LIN {X 0,Y 365.987,Z 762.314,A -85,B 0,C 180,E1 17582.28,E2 17582.28} C_VEL
LIN {X 0,Y 362.465,Z 777.838,A -85,B 0,C 180,E1 17579.586,E2 17579.586} C_VEL
LIN {X 0,Y 359.456,Z 791.622,A -85,B 0,C 180,E1 17576.759,E2 17576.759} C_VEL
LIN {X 0,Y 356.962,Z 803.911,A -85,B 0,C 180,E1 17573.786,E2 17573.786} C_VEL
LIN {X 0,Y 354.994,Z 814.892,A -85,B 0,C 180,E1 17570.612,E2 17570.612} C_VEL
LIN {X 0,Y 353.626,Z 823.927,A -85,B 0,C 180,E1 17567.438,E2 17567.438} C_VEL
LIN {X 0,Y 352.73,Z 831.669,A -85,B 0,C 180,E1 17564.108,E2 17564.108} C_VEL
LIN {X 0,Y 352.306,Z 837.449,A -85,B 0,C 180,E1 17560.895,E2 17560.895} C_VEL
LIN {X 0,Y 352.156,Z 841.876,A -85,B 0,C 180,E1 17557.503,E2 17557.503} C_VEL
LIN {X 0,Y 352.166,Z 844.497,A -85,B 0,C 180,E1 17554.395,E2 17554.395} C_VEL
LIN {X 0,Y 352.213,Z 845.642,A -85,B 0,C 180,E1 17551.137,E2 17551.137} C_VEL
LIN {X 0,Y 352.217,Z 845.355,A -85,B 0,C 180,E1 17548.046,E2 17548.046} C_VEL
LIN {X 0,Y 352.206,Z 843.421,A -85,B 0,C 180,E1 17544.786,E2 17544.786} C_VEL
LIN {X 0,Y 352.225,Z 839.976,A -85,B 0,C 180,E1 17541.51,E2 17541.51} C_VEL
LIN {X 0,Y 352.423,Z 835.044,A -85,B 0,C 180,E1 17538.378,E2 17538.378} C_VEL
LIN {X 0,Y 352.934,Z 828.184,A -85,B 0,C 180,E1 17535.031,E2 17535.031} C_VEL
LIN {X 0,Y 353.839,Z 820.007,A -85,B 0,C 180,E1 17531.889,E2 17531.889} C_VEL
LIN {X 0,Y 355.279,Z 809.812,A -85,B 0,C 180,E1 17528.677,E2 17528.677} C_VEL
LIN {X 0,Y 357.273,Z 797.828,A -85,B 0,C 180,E1 17525.53,E2 17525.53} C_VEL
LIN {X 0,Y 359.648,Z 784.987,A -85,B 0,C 180,E1 17522.694,E2 17522.694} C_VEL
LIN {X 0,Y 362.722,Z 769.51,A -85,B 0,C 180,E1 17519.795,E2 17519.795} C_VEL
LIN {X 0,Y 366.339,Z 752.001,A -85,B 0,C 180,E1 17517.031,E2 17517.031} C_VEL
LIN {X 0,Y 369.994,Z 734.378,A -85,B 0,C 180,E1 17514.667,E2 17514.667} C_VEL
LIN {X 0,Y 373.861,Z 715.366,A -85,B 0,C 180,E1 17512.523,E2 17512.523} C_VEL
LIN {X 0,Y 377.906,Z 695.003,A -85,B 0,C 180,E1 17510.58,E2 17510.58} C_VEL
LIN {X 0,Y 382.09,Z 673.141,A -85,B 0,C 180,E1 17508.841,E2 17508.841} C_VEL
LIN {X 0,Y 386.129,Z 650.609,A -85,B 0,C 180,E1 17507.368,E2 17507.368} C_VEL
LIN {X 0,Y 390.147,Z 626.368,A -85,B 0,C 180,E1 17506.112,E2 17506.112} C_VEL
LIN {X 0,Y 393.895,Z 600.938,A -85,B 0,C 180,E1 17505.107,E2 17505.107} C_VEL
LIN {X 0,Y 396.97,Z 573.317,A -85,B 0,C 180,E1 17504.265,E2 17504.265} C_VEL
LIN {X 0,Y 403.928,Z 504.871,A -85,B 0,C 180,E1 17502.414,E2 17502.414} C_VEL
LIN {X 0,Y 412.99,Z 436.759,A -85,B 0,C 180,E1 17500.479,E2 17500.479} C_VEL
LIN {X 0,Y 424.745,Z 366.791,A -85,B 0,C 180,E1 17498.462,E2 17498.462} C_VEL
LIN {X 0,Y 426.24,Z 358.784,A -85,B 0,C 180,E1 17498.201,E2 17498.201} C_VEL
LIN {X 0,Y 426.55,Z 354.223,A -85,B 0,C 180,E1 17497.156,E2 17497.156} C_VEL
LIN {X 0,Y 427.054,Z 351.949,A -85,B 0,C 180,E1 17496.325,E2 17496.325} C_VEL
LIN {X 0,Y 427.299,Z 351.738,A -85,B 0,C 180,E1 17495.886,E2 17495.886} C_VEL
LIN {X 0,Y 427.284,Z 352.228,A -85,B 0,C 180,E1 17495.743,E2 17495.743} C_VEL
LIN {X 0,Y 415.748,Z 415.551,A -85,B 0,C 180,E1 17493.926,E2 17493.926} C_VEL
LIN {X 0,Y 406.562,Z 477.379,A -85,B 0,C 180,E1 17492.151,E2 17492.151} C_VEL
LIN {X 0,Y 399.106,Z 542.752,A -85,B 0,C 180,E1 17490.336,E2 17490.336} C_VEL
LIN {X 0,Y 396.477,Z 567.509,A -85,B 0,C 180,E1 17489.494,E2 17489.494} C_VEL
LIN {X 0,Y 393.293,Z 591.201,A -85,B 0,C 180,E1 17488.387,E2 17488.387} C_VEL
LIN {X 0,Y 389.623,Z 613.913,A -85,B 0,C 180,E1 17487.016,E2 17487.016} C_VEL
LIN {X 0,Y 385.453,Z 636.079,A -85,B 0,C 180,E1 17485.343,E2 17485.343} C_VEL
LIN {X 0,Y 381.122,Z 656.641,A -85,B 0,C 180,E1 17483.421,E2 17483.421} C_VEL
LIN {X 0,Y 376.79,Z 675.215,A -85,B 0,C 180,E1 17481.32,E2 17481.32} C_VEL
LIN {X 0,Y 372.567,Z 692.109,A -85,B 0,C 180,E1 17479.032,E2 17479.032} C_VEL
LIN {X 0,Y 368.567,Z 707.5,A -85,B 0,C 180,E1 17476.551,E2 17476.551} C_VEL
LIN {X 0,Y 364.962,Z 721.167,A -85,B 0,C 180,E1 17473.953,E2 17473.953} C_VEL
LIN {X 0,Y 361.517,Z 734.047,A -85,B 0,C 180,E1 17471.003,E2 17471.003} C_VEL
LIN {X 0,Y 358.694,Z 744.9,A -85,B 0,C 180,E1 17468.014,E2 17468.014} C_VEL
LIN {X 0,Y 356.397,Z 754.518,A -85,B 0,C 180,E1 17464.83,E2 17464.83} C_VEL
LIN {X 0,Y 354.639,Z 762.753,A -85,B 0,C 180,E1 17461.456,E2 17461.456} C_VEL
LIN {X 0,Y 353.45,Z 769.171,A -85,B 0,C 180,E1 17458.057,E2 17458.057} C_VEL
LIN {X 0,Y 352.739,Z 774.193,A -85,B 0,C 180,E1 17454.472,E2 17454.472} C_VEL
LIN {X 0,Y 352.395,Z 777.476,A -85,B 0,C 180,E1 17451.025,E2 17451.025} C_VEL
LIN {X 0,Y 352.253,Z 779.104,A -85,B 0,C 180,E1 17447.711,E2 17447.711} C_VEL
LIN {X 0,Y 352.227,Z 779.342,A -85,B 0,C 180,E1 17444.223,E2 17444.223} C_VEL
LIN {X 0,Y 352.257,Z 778.2,A -85,B 0,C 180,E1 17440.946,E2 17440.946} C_VEL
LIN {X 0,Y 352.388,Z 775.578,A -85,B 0,C 180,E1 17437.656,E2 17437.656} C_VEL
LIN {X 0,Y 352.757,Z 771.52,A -85,B 0,C 180,E1 17434.303,E2 17434.303} C_VEL
LIN {X 0,Y 353.475,Z 765.83,A -85,B 0,C 180,E1 17430.935,E2 17430.935} C_VEL
LIN {X 0,Y 354.654,Z 758.568,A -85,B 0,C 180,E1 17427.615,E2 17427.615} C_VEL
LIN {X 0,Y 356.419,Z 749.576,A -85,B 0,C 180,E1 17424.307,E2 17424.307} C_VEL
LIN {X 0,Y 358.837,Z 738.627,A -85,B 0,C 180,E1 17421.025,E2 17421.025} C_VEL
LIN {X 0,Y 361.659,Z 726.557,A -85,B 0,C 180,E1 17418.048,E2 17418.048} C_VEL
LIN {X 0,Y 365.008,Z 712.783,A -85,B 0,C 180,E1 17415.193,E2 17415.193} C_VEL
LIN {X 0,Y 368.625,Z 698.003,A -85,B 0,C 180,E1 17412.603,E2 17412.603} C_VEL
LIN {X 0,Y 372.462,Z 681.884,A -85,B 0,C 180,E1 17410.231,E2 17410.231} C_VEL
LIN {X 0,Y 376.443,Z 664.226,A -85,B 0,C 180,E1 17408.041,E2 17408.041} C_VEL
LIN {X 0,Y 380.473,Z 645.175,A -85,B 0,C 180,E1 17406.063,E2 17406.063} C_VEL
LIN {X 0,Y 384.229,Z 625.745,A -85,B 0,C 180,E1 17404.382,E2 17404.382} C_VEL
LIN {X 0,Y 387.547,Z 605.931,A -85,B 0,C 180,E1 17402.983,E2 17402.983} C_VEL
LIN {X 0,Y 390.527,Z 585.074,A -85,B 0,C 180,E1 17401.793,E2 17401.793} C_VEL
LIN {X 0,Y 393.119,Z 563.144,A -85,B 0,C 180,E1 17400.816,E2 17400.816} C_VEL
LIN {X 0,Y 395.064,Z 541.461,A -85,B 0,C 180,E1 17400.105,E2 17400.105} C_VEL
LIN {X 0,Y 397.486,Z 497.686,A -85,B 0,C 180,E1 17399.14,E2 17399.14} C_VEL
LIN {X 0,Y 405.981,Z 342.64,A -85,B 0,C 180,E1 17395.845,E2 17395.845} C_VEL
LIN {X 0,Y 392.058,Z 321.721,A -85,B 0,C 180,E1 17393.047,E2 17393.047} C_VEL
LIN {X 0,Y 379.817,Z 304.351,A -85,B 0,C 180,E1 17390.335,E2 17390.335} C_VEL
LIN {X 0,Y 369.449,Z 290.34,A -85,B 0,C 180,E1 17387.849,E2 17387.849} C_VEL
LIN {X 0,Y 365.575,Z 285.201,A -85,B 0,C 180,E1 17386.854,E2 17386.854} C_VEL
LIN {X 0,Y 362.474,Z 280.851,A -85,B 0,C 180,E1 17386.034,E2 17386.034} C_VEL
LIN {X 0,Y 358.985,Z 276.815,A -85,B 0,C 180,E1 17385.117,E2 17385.117} C_VEL
LIN {X 0,Y 357.684,Z 274.526,A -85,B 0,C 180,E1 17384.73,E2 17384.73} C_VEL
LIN {X 0,Y 355.038,Z 271.984,A -85,B 0,C 180,E1 17384.017,E2 17384.017} C_VEL
LIN {X 0,Y 353.876,Z 268.895,A -85,B 0,C 180,E1 17383.606,E2 17383.606} C_VEL
LIN {X 0,Y 353.84,Z 268.66,A -85,B 0,C 180,E1 17379.557,E2 17379.557} C_VEL
LIN {X 0,Y 353.836,Z 268.649,A -85,B 0,C 180,E1 17375.515,E2 17375.515} C_VEL
LIN {X 0,Y 353.842,Z 268.652,A -85,B 0,C 180,E1 17371.297,E2 17371.297} C_VEL
LIN {X 0,Y 353.839,Z 268.655,A -85,B 0,C 180,E1 17367.248,E2 17367.248} C_VEL
LIN {X 0,Y 353.825,Z 268.656,A -85,B 0,C 180,E1 17363.609,E2 17363.609} C_VEL
LIN {X 0,Y 352.854,Z 268.776,A -85,B 0,C 180,E1 17362.362,E2 17362.362} C_VEL
LIN {X 0,Y 348.27,Z 269.351,A -85,B 0,C 180,E1 17360.005,E2 17360.005} C_VEL
LIN {X 0,Y 346.039,Z 269.618,A -85,B 0,C 180,E1 17358.378,E2 17358.378} C_VEL
LIN {X 0,Y 345.889,Z 269.637,A -85,B 0,C 180,E1 17357.915,E2 17357.915} C_VEL
LIN {X 0,Y 345.884,Z 269.641,A -85,B 0,C 180,E1 17353.67,E2 17353.67} C_VEL
LIN {X 0,Y 345.884,Z 269.643,A -85,B 0,C 180,E1 17349.351,E2 17349.351} C_VEL
LIN {X 0,Y 345.884,Z 269.643,A -85,B 0,C 180,E1 17345.18,E2 17345.18} C_VEL
LIN {X 0,Y 345.882,Z 269.642,A -85,B 0,C 180,E1 17341.137,E2 17341.137} C_VEL
LIN {X 0,Y 345.885,Z 269.64,A -85,B 0,C 180,E1 17336.956,E2 17336.956} C_VEL
LIN {X 0,Y 345.885,Z 269.639,A -85,B 0,C 180,E1 17332.834,E2 17332.834} C_VEL
LIN {X 0,Y 345.887,Z 269.642,A -85,B 0,C 180,E1 17328.723,E2 17328.723} C_VEL
LIN {X 0,Y 345.888,Z 269.645,A -85,B 0,C 180,E1 17324.618,E2 17324.618} C_VEL
LIN {X 0,Y 345.901,Z 269.645,A -85,B 0,C 180,E1 17320.349,E2 17320.349} C_VEL
LIN {X 0,Y 345.903,Z 269.647,A -85,B 0,C 180,E1 17316.13,E2 17316.13} C_VEL
LIN {X 0,Y 345.9,Z 269.648,A -85,B 0,C 180,E1 17311.811,E2 17311.811} C_VEL
LIN {X 0,Y 345.902,Z 269.65,A -85,B 0,C 180,E1 17307.732,E2 17307.732} C_VEL
LIN {X 0,Y 345.886,Z 269.652,A -85,B 0,C 180,E1 17303.508,E2 17303.508} C_VEL
LIN {X 0,Y 345.883,Z 269.651,A -85,B 0,C 180,E1 17299.414,E2 17299.414} C_VEL
LIN {X 0,Y 345.875,Z 269.649,A -85,B 0,C 180,E1 17295.249,E2 17295.249} C_VEL
LIN {X 0,Y 345.87,Z 269.645,A -85,B 0,C 180,E1 17291.165,E2 17291.165} C_VEL
LIN {X 0,Y 345.861,Z 269.646,A -85,B 0,C 180,E1 17286.972,E2 17286.972} C_VEL
LIN {X 0,Y 345.859,Z 269.653,A -85,B 0,C 180,E1 17282.815,E2 17282.815} C_VEL
LIN {X 0,Y 345.856,Z 269.654,A -85,B 0,C 180,E1 17278.507,E2 17278.507} C_VEL
LIN {X 0,Y 345.859,Z 269.645,A -85,B 0,C 180,E1 17274.357,E2 17274.357} C_VEL
LIN {X 0,Y 345.863,Z 269.654,A -85,B 0,C 180,E1 17270.177,E2 17270.177} C_VEL
LIN {X 0,Y 345.869,Z 269.645,A -85,B 0,C 180,E1 17265.944,E2 17265.944} C_VEL
LIN {X 0,Y 345.874,Z 269.647,A -85,B 0,C 180,E1 17261.806,E2 17261.806} C_VEL
LIN {X 0,Y 345.88,Z 269.65,A -85,B 0,C 180,E1 17257.669,E2 17257.669} C_VEL
LIN {X 0,Y 345.94,Z 269.93,A -85,B 0,C 180,E1 17257.391,E2 17257.391} C_VEL
LIN {X 0,Y 347.396,Z 273.438,A -85,B 0,C 180,E1 17256.416,E2 17256.416} C_VEL
LIN {X 0,Y 348.675,Z 275.305,A -85,B 0,C 180,E1 17255.789,E2 17255.789} C_VEL
LIN {X 0,Y 350.72,Z 279.095,A -85,B 0,C 180,E1 17254.681,E2 17254.681} C_VEL
LIN {X 0,Y 354.332,Z 286.186,A -85,B 0,C 180,E1 17252.727,E2 17252.727} C_VEL
LIN {X 0,Y 360.76,Z 295.311,A -85,B 0,C 180,E1 17250.803,E2 17250.803} C_VEL
LIN {X 0,Y 373.143,Z 313.414,A -85,B 0,C 180,E1 17247.524,E2 17247.524} C_VEL
LIN {X 0,Y 384.602,Z 331.118,A -85,B 0,C 180,E1 17244.772,E2 17244.772} C_VEL
LIN {X 0,Y 397.375,Z 351.926,A -85,B 0,C 180,E1 17241.964,E2 17241.964} C_VEL
LIN {X 0,Y 402.124,Z 360.571,A -85,B 0,C 180,E1 17240.95,E2 17240.95} C_VEL
LIN {X 0,Y 390.839,Z 551.737,A -85,B 0,C 180,E1 17236.825,E2 17236.825} C_VEL
LIN {X 0,Y 387.902,Z 601.626,A -85,B 0,C 180,E1 17235.696,E2 17235.696} C_VEL
LIN {X 0,Y 385.427,Z 624.723,A -85,B 0,C 180,E1 17234.955,E2 17234.955} C_VEL
LIN {X 0,Y 382.332,Z 646.717,A -85,B 0,C 180,E1 17233.981,E2 17233.981} C_VEL
LIN {X 0,Y 378.753,Z 668.624,A -85,B 0,C 180,E1 17232.72,E2 17232.72} C_VEL
LIN {X 0,Y 374.834,Z 689.594,A -85,B 0,C 180,E1 17231.211,E2 17231.211} C_VEL
LIN {X 0,Y 370.706,Z 709.59,A -85,B 0,C 180,E1 17229.456,E2 17229.456} C_VEL
LIN {X 0,Y 366.414,Z 728.906,A -85,B 0,C 180,E1 17227.391,E2 17227.391} C_VEL
LIN {X 0,Y 362.411,Z 746.037,A -85,B 0,C 180,E1 17225.21,E2 17225.21} C_VEL
LIN {X 0,Y 358.517,Z 762.431,A -85,B 0,C 180,E1 17222.752,E2 17222.752} C_VEL
LIN {X 0,Y 354.962,Z 777.449,A -85,B 0,C 180,E1 17220.09,E2 17220.09} C_VEL
LIN {X 0,Y 351.773,Z 791.358,A -85,B 0,C 180,E1 17217.168,E2 17217.168} C_VEL
LIN {X 0,Y 349.042,Z 804.226,A -85,B 0,C 180,E1 17213.962,E2 17213.962} C_VEL
LIN {X 0,Y 347.041,Z 815.018,A -85,B 0,C 180,E1 17210.753,E2 17210.753} C_VEL
LIN {X 0,Y 345.579,Z 824.337,A -85,B 0,C 180,E1 17207.336,E2 17207.336} C_VEL
LIN {X 0,Y 344.698,Z 831.806,A -85,B 0,C 180,E1 17203.929,E2 17203.929} C_VEL
LIN {X 0,Y 344.289,Z 837.602,A -85,B 0,C 180,E1 17200.54,E2 17200.54} C_VEL
LIN {X 0,Y 344.183,Z 841.606,A -85,B 0,C 180,E1 17197.174,E2 17197.174} C_VEL
LIN {X 0,Y 344.204,Z 844.093,A -85,B 0,C 180,E1 17193.829,E2 17193.829} C_VEL
LIN {X 0,Y 344.25,Z 844.918,A -85,B 0,C 180,E1 17190.83,E2 17190.83} C_VEL
LIN {X 0,Y 344.248,Z 844.467,A -85,B 0,C 180,E1 17187.64,E2 17187.64} C_VEL
LIN {X 0,Y 344.231,Z 842.486,A -85,B 0,C 180,E1 17184.498,E2 17184.498} C_VEL
LIN {X 0,Y 344.252,Z 838.914,A -85,B 0,C 180,E1 17181.143,E2 17181.143} C_VEL
LIN {X 0,Y 344.481,Z 833.899,A -85,B 0,C 180,E1 17177.936,E2 17177.936} C_VEL
LIN {X 0,Y 345.05,Z 826.928,A -85,B 0,C 180,E1 17174.537,E2 17174.537} C_VEL
LIN {X 0,Y 346.051,Z 818.588,A -85,B 0,C 180,E1 17171.292,E2 17171.292} C_VEL
LIN {X 0,Y 347.606,Z 808.312,A -85,B 0,C 180,E1 17168.04,E2 17168.04} C_VEL
LIN {X 0,Y 349.803,Z 796.062,A -85,B 0,C 180,E1 17164.791,E2 17164.791} C_VEL
LIN {X 0,Y 352.544,Z 782.277,A -85,B 0,C 180,E1 17161.728,E2 17161.728} C_VEL
LIN {X 0,Y 355.894,Z 766.369,A -85,B 0,C 180,E1 17158.763,E2 17158.763} C_VEL
LIN {X 0,Y 359.691,Z 748.99,A -85,B 0,C 180,E1 17156.03,E2 17156.03} C_VEL
LIN {X 0,Y 363.773,Z 730.564,A -85,B 0,C 180,E1 17153.579,E2 17153.579} C_VEL
LIN {X 0,Y 367.934,Z 711.368,A -85,B 0,C 180,E1 17151.414,E2 17151.414} C_VEL
LIN {X 0,Y 372.301,Z 690.641,A -85,B 0,C 180,E1 17149.463,E2 17149.463} C_VEL
LIN {X 0,Y 376.777,Z 668.441,A -85,B 0,C 180,E1 17147.722,E2 17147.722} C_VEL
LIN {X 0,Y 381.333,Z 644.505,A -85,B 0,C 180,E1 17146.193,E2 17146.193} C_VEL
LIN {X 0,Y 385.584,Z 620.731,A -85,B 0,C 180,E1 17144.998,E2 17144.998} C_VEL
LIN {X 0,Y 389.51,Z 595.619,A -85,B 0,C 180,E1 17144.014,E2 17144.014} C_VEL
LIN {X 0,Y 392.91,Z 567.261,A -85,B 0,C 180,E1 17143.15,E2 17143.15} C_VEL
LIN {X 0,Y 400.496,Z 503.181,A -85,B 0,C 180,E1 17141.343,E2 17141.343} C_VEL
LIN {X 0,Y 410.231,Z 439.062,A -85,B 0,C 180,E1 17139.47,E2 17139.47} C_VEL
LIN {X 0,Y 422.676,Z 372.581,A -85,B 0,C 180,E1 17137.534,E2 17137.534} C_VEL
LIN {X 0,Y 424.558,Z 363.407,A -85,B 0,C 180,E1 17137.248,E2 17137.248} C_VEL
LIN {X 0,Y 424.992,Z 361.112,A -85,B 0,C 180,E1 17136.587,E2 17136.587} C_VEL
LIN {X 0,Y 411.882,Z 427.07,A -85,B 0,C 180,E1 17134.679,E2 17134.679} C_VEL
LIN {X 0,Y 401.559,Z 490.527,A -85,B 0,C 180,E1 17132.823,E2 17132.823} C_VEL
LIN {X 0,Y 393.413,Z 555.583,A -85,B 0,C 180,E1 17130.917,E2 17130.917} C_VEL
LIN {X 0,Y 390.393,Z 578.397,A -85,B 0,C 180,E1 17129.985,E2 17129.985} C_VEL
LIN {X 0,Y 386.887,Z 600.317,A -85,B 0,C 180,E1 17128.823,E2 17128.823} C_VEL
LIN {X 0,Y 382.842,Z 622.167,A -85,B 0,C 180,E1 17127.366,E2 17127.366} C_VEL
LIN {X 0,Y 378.512,Z 642.8,A -85,B 0,C 180,E1 17125.673,E2 17125.673} C_VEL
LIN {X 0,Y 373.851,Z 662.951,A -85,B 0,C 180,E1 17123.653,E2 17123.653} C_VEL
LIN {X 0,Y 369.383,Z 680.694,A -85,B 0,C 180,E1 17121.519,E2 17121.519} C_VEL
LIN {X 0,Y 365.071,Z 696.933,A -85,B 0,C 180,E1 17119.189,E2 17119.189} C_VEL
LIN {X 0,Y 360.573,Z 712.928,A -85,B 0,C 180,E1 17116.432,E2 17116.432} C_VEL
LIN {X 0,Y 356.695,Z 726.498,A -85,B 0,C 180,E1 17113.621,E2 17113.621} C_VEL
LIN {X 0,Y 353.249,Z 738.694,A -85,B 0,C 180,E1 17110.604,E2 17110.604} C_VEL
LIN {X 0,Y 350.468,Z 749.046,A -85,B 0,C 180,E1 17107.543,E2 17107.543} C_VEL
LIN {X 0,Y 348.085,Z 758.409,A -85,B 0,C 180,E1 17104.12,E2 17104.12} C_VEL
LIN {X 0,Y 346.47,Z 765.632,A -85,B 0,C 180,E1 17100.829,E2 17100.829} C_VEL
LIN {X 0,Y 345.355,Z 771.623,A -85,B 0,C 180,E1 17097.347,E2 17097.347} C_VEL
LIN {X 0,Y 344.742,Z 775.801,A -85,B 0,C 180,E1 17094.009,E2 17094.009} C_VEL
LIN {X 0,Y 344.403,Z 778.691,A -85,B 0,C 180,E1 17090.477,E2 17090.477} C_VEL
LIN {X 0,Y 344.29,Z 780.105,A -85,B 0,C 180,E1 17087.081,E2 17087.081} C_VEL
LIN {X 0,Y 344.261,Z 780.013,A -85,B 0,C 180,E1 17083.813,E2 17083.813} C_VEL
LIN {X 0,Y 344.305,Z 778.571,A -85,B 0,C 180,E1 17080.317,E2 17080.317} C_VEL
LIN {X 0,Y 344.481,Z 775.704,A -85,B 0,C 180,E1 17076.934,E2 17076.934} C_VEL
LIN {X 0,Y 344.938,Z 771.274,A -85,B 0,C 180,E1 17073.491,E2 17073.491} C_VEL
LIN {X 0,Y 345.82,Z 765.205,A -85,B 0,C 180,E1 17069.991,E2 17069.991} C_VEL
LIN {X 0,Y 347.182,Z 757.638,A -85,B 0,C 180,E1 17066.632,E2 17066.632} C_VEL
LIN {X 0,Y 349.181,Z 748.138,A -85,B 0,C 180,E1 17063.244,E2 17063.244} C_VEL
LIN {X 0,Y 351.752,Z 737.194,A -85,B 0,C 180,E1 17060.032,E2 17060.032} C_VEL
LIN {X 0,Y 354.833,Z 724.842,A -85,B 0,C 180,E1 17057.011,E2 17057.011} C_VEL
LIN {X 0,Y 358.34,Z 710.978,A -85,B 0,C 180,E1 17054.189,E2 17054.189} C_VEL
LIN {X 0,Y 362.357,Z 695.125,A -85,B 0,C 180,E1 17051.472,E2 17051.472} C_VEL
LIN {X 0,Y 366.442,Z 678.508,A -85,B 0,C 180,E1 17049.073,E2 17049.073} C_VEL
LIN {X 0,Y 370.596,Z 660.697,A -85,B 0,C 180,E1 17046.92,E2 17046.92} C_VEL
LIN {X 0,Y 374.617,Z 641.776,A -85,B 0,C 180,E1 17045.02,E2 17045.02} C_VEL
LIN {X 0,Y 378.498,Z 621.527,A -85,B 0,C 180,E1 17043.331,E2 17043.331} C_VEL
LIN {X 0,Y 382.017,Z 600.736,A -85,B 0,C 180,E1 17041.919,E2 17041.919} C_VEL
LIN {X 0,Y 385.086,Z 579.227,A -85,B 0,C 180,E1 17040.754,E2 17040.754} C_VEL
LIN {X 0,Y 387.482,Z 557.645,A -85,B 0,C 180,E1 17039.863,E2 17039.863} C_VEL
LIN {X 0,Y 389.383,Z 534.657,A -85,B 0,C 180,E1 17039.177,E2 17039.177} C_VEL
LIN {X 0,Y 400.255,Z 346.403,A -85,B 0,C 180,E1 17035.121,E2 17035.121} C_VEL
LIN {X 0,Y 386.989,Z 326.388,A -85,B 0,C 180,E1 17032.374,E2 17032.374} C_VEL
LIN {X 0,Y 373.822,Z 307.654,A -85,B 0,C 180,E1 17029.371,E2 17029.371} C_VEL
LIN {X 0,Y 364.84,Z 295.625,A -85,B 0,C 180,E1 17027.135,E2 17027.135} C_VEL
LIN {X 0,Y 361.47,Z 291.189,A -85,B 0,C 180,E1 17026.266,E2 17026.266} C_VEL
LIN {X 0,Y 358.052,Z 286.587,A -85,B 0,C 180,E1 17025.344,E2 17025.344} C_VEL
LIN {X 0,Y 354.901,Z 282.379,A -85,B 0,C 180,E1 17024.46,E2 17024.46} C_VEL
LIN {X 0,Y 353.664,Z 280.894,A -85,B 0,C 180,E1 17024.111,E2 17024.111} C_VEL
LIN {X 0,Y 350.862,Z 277.341,A -85,B 0,C 180,E1 17023.305,E2 17023.305} C_VEL
LIN {X 0,Y 349.902,Z 275.6,A -85,B 0,C 180,E1 17023.003,E2 17023.003} C_VEL
LIN {X 0,Y 347.122,Z 273.01,A -85,B 0,C 180,E1 17022.224,E2 17022.224} C_VEL
LIN {X 0,Y 345.934,Z 269.916,A -85,B 0,C 180,E1 17021.78,E2 17021.78} C_VEL
LIN {X 0,Y 345.904,Z 269.641,A -85,B 0,C 180,E1 17021.506,E2 17021.506} C_VEL
LIN {X 0,Y 345.909,Z 269.644,A -85,B 0,C 180,E1 17017.308,E2 17017.308} C_VEL
LIN {X 0,Y 345.91,Z 269.639,A -85,B 0,C 180,E1 17013.15,E2 17013.15} C_VEL
LIN {X 0,Y 345.918,Z 269.631,A -85,B 0,C 180,E1 17009.008,E2 17009.008} C_VEL
LIN {X 0,Y 345.92,Z 269.633,A -85,B 0,C 180,E1 17004.695,E2 17004.695} C_VEL
LIN {X 0,Y 345.917,Z 269.641,A -85,B 0,C 180,E1 17000.519,E2 17000.519} C_VEL
LIN {X 0,Y 345.889,Z 269.637,A -85,B 0,C 180,E1 16997.915,E2 16997.915} C_VEL
LIN {X 0,Y 344.898,Z 269.771,A -85,B 0,C 180,E1 16996.639,E2 16996.639} C_VEL
LIN {X 0,Y 340.177,Z 270.369,A -85,B 0,C 180,E1 16994.136,E2 16994.136} C_VEL
LIN {X 0,Y 338.068,Z 270.627,A -85,B 0,C 180,E1 16992.467,E2 16992.467} C_VEL
LIN {X 0,Y 337.961,Z 270.637,A -85,B 0,C 180,E1 16992.087,E2 16992.087} C_VEL
LIN {X 0,Y 337.947,Z 270.638,A -85,B 0,C 180,E1 16987.818,E2 16987.818} C_VEL
LIN {X 0,Y 337.945,Z 270.639,A -85,B 0,C 180,E1 16983.656,E2 16983.656} C_VEL
LIN {X 0,Y 337.941,Z 270.641,A -85,B 0,C 180,E1 16979.412,E2 16979.412} C_VEL
LIN {X 0,Y 337.938,Z 270.643,A -85,B 0,C 180,E1 16975.181,E2 16975.181} C_VEL
LIN {X 0,Y 337.942,Z 270.643,A -85,B 0,C 180,E1 16970.938,E2 16970.938} C_VEL
LIN {X 0,Y 337.947,Z 270.642,A -85,B 0,C 180,E1 16966.699,E2 16966.699} C_VEL
LIN {X 0,Y 337.959,Z 270.638,A -85,B 0,C 180,E1 16962.414,E2 16962.414} C_VEL
LIN {X 0,Y 337.971,Z 270.632,A -85,B 0,C 180,E1 16958.103,E2 16958.103} C_VEL
LIN {X 0,Y 337.957,Z 270.631,A -85,B 0,C 180,E1 16953.767,E2 16953.767} C_VEL
LIN {X 0,Y 337.951,Z 270.628,A -85,B 0,C 180,E1 16949.566,E2 16949.566} C_VEL
LIN {X 0,Y 337.94,Z 270.627,A -85,B 0,C 180,E1 16945.402,E2 16945.402} C_VEL
LIN {X 0,Y 337.93,Z 270.633,A -85,B 0,C 180,E1 16941.157,E2 16941.157} C_VEL
LIN {X 0,Y 337.923,Z 270.639,A -85,B 0,C 180,E1 16936.853,E2 16936.853} C_VEL
LIN {X 0,Y 337.921,Z 270.642,A -85,B 0,C 180,E1 16932.471,E2 16932.471} C_VEL
LIN {X 0,Y 337.929,Z 270.642,A -85,B 0,C 180,E1 16928.162,E2 16928.162} C_VEL
LIN {X 0,Y 337.937,Z 270.634,A -85,B 0,C 180,E1 16923.9,E2 16923.9} C_VEL
LIN {X 0,Y 337.955,Z 270.634,A -85,B 0,C 180,E1 16919.659,E2 16919.659} C_VEL
LIN {X 0,Y 337.953,Z 270.636,A -85,B 0,C 180,E1 16915.416,E2 16915.416} C_VEL
LIN {X 0,Y 337.951,Z 270.633,A -85,B 0,C 180,E1 16911.148,E2 16911.148} C_VEL
LIN {X 0,Y 337.938,Z 270.636,A -85,B 0,C 180,E1 16906.829,E2 16906.829} C_VEL
LIN {X 0,Y 337.941,Z 270.636,A -85,B 0,C 180,E1 16902.788,E2 16902.788} C_VEL
LIN {X 0,Y 337.994,Z 270.844,A -85,B 0,C 180,E1 16899.296,E2 16899.296} C_VEL
LIN {X 0,Y 339.206,Z 274.076,A -85,B 0,C 180,E1 16898.378,E2 16898.378} C_VEL
LIN {X 0,Y 340.793,Z 276.266,A -85,B 0,C 180,E1 16897.577,E2 16897.577} C_VEL
LIN {X 0,Y 342.723,Z 280.006,A -85,B 0,C 180,E1 16896.44,E2 16896.44} C_VEL
LIN {X 0,Y 346.275,Z 286.469,A -85,B 0,C 180,E1 16894.562,E2 16894.562} C_VEL
LIN {X 0,Y 357.277,Z 301.929,A -85,B 0,C 180,E1 16891.27,E2 16891.27} C_VEL
LIN {X 0,Y 369.538,Z 319.979,A -85,B 0,C 180,E1 16887.972,E2 16887.972} C_VEL
LIN {X 0,Y 380.777,Z 337.544,A -85,B 0,C 180,E1 16885.216,E2 16885.216} C_VEL
LIN {X 0,Y 393.502,Z 358.5,A -85,B 0,C 180,E1 16882.353,E2 16882.353} C_VEL
LIN {X 0,Y 396.438,Z 364.045,A -85,B 0,C 180,E1 16881.718,E2 16881.718} C_VEL
LIN {X 0,Y 384.093,Z 563.816,A -85,B 0,C 180,E1 16877.334,E2 16877.334} C_VEL
LIN {X 0,Y 381.685,Z 601.896,A -85,B 0,C 180,E1 16876.444,E2 16876.444} C_VEL
LIN {X 0,Y 379.098,Z 624.989,A -85,B 0,C 180,E1 16875.688,E2 16875.688} C_VEL
LIN {X 0,Y 375.798,Z 647.424,A -85,B 0,C 180,E1 16874.671,E2 16874.671} C_VEL
LIN {X 0,Y 372.225,Z 668.32,A -85,B 0,C 180,E1 16873.442,E2 16873.442} C_VEL
LIN {X 0,Y 368.156,Z 689.258,A -85,B 0,C 180,E1 16871.913,E2 16871.913} C_VEL
LIN {X 0,Y 363.84,Z 709.358,A -85,B 0,C 180,E1 16870.12,E2 16870.12} C_VEL
LIN {X 0,Y 359.49,Z 728.135,A -85,B 0,C 180,E1 16868.082,E2 16868.082} C_VEL
LIN {X 0,Y 355.26,Z 745.584,A -85,B 0,C 180,E1 16865.829,E2 16865.829} C_VEL
LIN {X 0,Y 351.195,Z 762.007,A -85,B 0,C 180,E1 16863.328,E2 16863.328} C_VEL
LIN {X 0,Y 347.489,Z 777.06,A -85,B 0,C 180,E1 16860.615,E2 16860.615} C_VEL
LIN {X 0,Y 344.205,Z 790.676,A -85,B 0,C 180,E1 16857.693,E2 16857.693} C_VEL
LIN {X 0,Y 341.312,Z 803.635,A -85,B 0,C 180,E1 16854.395,E2 16854.395} C_VEL
LIN {X 0,Y 339.182,Z 814.526,A -85,B 0,C 180,E1 16851.076,E2 16851.076} C_VEL
LIN {X 0,Y 337.705,Z 823.408,A -85,B 0,C 180,E1 16847.754,E2 16847.754} C_VEL
LIN {X 0,Y 336.729,Z 831.28,A -85,B 0,C 180,E1 16844.09,E2 16844.09} C_VEL
LIN {X 0,Y 336.307,Z 837.033,A -85,B 0,C 180,E1 16840.62,E2 16840.62} C_VEL
LIN {X 0,Y 336.202,Z 840.827,A -85,B 0,C 180,E1 16837.345,E2 16837.345} C_VEL
LIN {X 0,Y 336.235,Z 843.336,A -85,B 0,C 180,E1 16833.92,E2 16833.92} C_VEL
LIN {X 0,Y 336.287,Z 844.155,A -85,B 0,C 180,E1 16830.85,E2 16830.85} C_VEL
LIN {X 0,Y 336.282,Z 843.715,A -85,B 0,C 180,E1 16827.613,E2 16827.613} C_VEL
LIN {X 0,Y 336.256,Z 841.706,A -85,B 0,C 180,E1 16824.367,E2 16824.367} C_VEL
LIN {X 0,Y 336.27,Z 838.34,A -85,B 0,C 180,E1 16821.104,E2 16821.104} C_VEL
LIN {X 0,Y 336.501,Z 833.336,A -85,B 0,C 180,E1 16817.82,E2 16817.82} C_VEL
LIN {X 0,Y 337.096,Z 826.457,A -85,B 0,C 180,E1 16814.339,E2 16814.339} C_VEL
LIN {X 0,Y 338.142,Z 818.115,A -85,B 0,C 180,E1 16811.017,E2 16811.017} C_VEL
LIN {X 0,Y 339.78,Z 807.945,A -85,B 0,C 180,E1 16807.689,E2 16807.689} C_VEL
LIN {X 0,Y 342.095,Z 795.767,A -85,B 0,C 180,E1 16804.368,E2 16804.368} C_VEL
LIN {X 0,Y 344.981,Z 782.035,A -85,B 0,C 180,E1 16801.24,E2 16801.24} C_VEL
LIN {X 0,Y 348.374,Z 766.797,A -85,B 0,C 180,E1 16798.315,E2 16798.315} C_VEL
LIN {X 0,Y 352.239,Z 750.241,A -85,B 0,C 180,E1 16795.605,E2 16795.605} C_VEL
LIN {X 0,Y 356.482,Z 732.277,A -85,B 0,C 180,E1 16793.113,E2 16793.113} C_VEL
LIN {X 0,Y 360.966,Z 712.766,A -85,B 0,C 180,E1 16790.834,E2 16790.834} C_VEL
LIN {X 0,Y 365.714,Z 691.846,A -85,B 0,C 180,E1 16788.783,E2 16788.783} C_VEL
LIN {X 0,Y 370.471,Z 670.123,A -85,B 0,C 180,E1 16787.005,E2 16787.005} C_VEL
LIN {X 0,Y 375.151,Z 647.777,A -85,B 0,C 180,E1 16785.495,E2 16785.495} C_VEL
LIN {X 0,Y 380.114,Z 622.631,A -85,B 0,C 180,E1 16784.155,E2 16784.155} C_VEL
LIN {X 0,Y 384.998,Z 594.61,A -85,B 0,C 180,E1 16783.009,E2 16783.009} C_VEL
LIN {X 0,Y 389.291,Z 562.75,A -85,B 0,C 180,E1 16782.012,E2 16782.012} C_VEL
LIN {X 0,Y 397.665,Z 502.064,A -85,B 0,C 180,E1 16780.233,E2 16780.233} C_VEL
LIN {X 0,Y 408.652,Z 438.65,A -85,B 0,C 180,E1 16778.347,E2 16778.347} C_VEL
LIN {X 0,Y 418.754,Z 389.396,A -85,B 0,C 180,E1 16776.895,E2 16776.895} C_VEL
LIN {X 0,Y 405.45,Z 453.865,A -85,B 0,C 180,E1 16775.007,E2 16775.007} C_VEL
LIN {X 0,Y 395.675,Z 511.235,A -85,B 0,C 180,E1 16773.304,E2 16773.304} C_VEL
LIN {X 0,Y 389.087,Z 558.891,A -85,B 0,C 180,E1 16771.834,E2 16771.834} C_VEL
LIN {X 0,Y 385.59,Z 581.894,A -85,B 0,C 180,E1 16770.84,E2 16770.84} C_VEL
LIN {X 0,Y 381.364,Z 605.259,A -85,B 0,C 180,E1 16769.533,E2 16769.533} C_VEL
LIN {X 0,Y 376.91,Z 626.822,A -85,B 0,C 180,E1 16768.006,E2 16768.006} C_VEL
LIN {X 0,Y 372.534,Z 645.783,A -85,B 0,C 180,E1 16766.373,E2 16766.373} C_VEL
LIN {X 0,Y 367.786,Z 664.767,A -85,B 0,C 180,E1 16764.409,E2 16764.409} C_VEL
LIN {X 0,Y 363.069,Z 682.253,A -85,B 0,C 180,E1 16762.253,E2 16762.253} C_VEL
LIN {X 0,Y 358.516,Z 698.33,A -85,B 0,C 180,E1 16759.893,E2 16759.893} C_VEL
LIN {X 0,Y 354.007,Z 713.355,A -85,B 0,C 180,E1 16757.253,E2 16757.253} C_VEL
LIN {X 0,Y 349.862,Z 726.978,A -85,B 0,C 180,E1 16754.399,E2 16754.399} C_VEL
LIN {X 0,Y 346.169,Z 739.222,A -85,B 0,C 180,E1 16751.329,E2 16751.329} C_VEL
LIN {X 0,Y 343.158,Z 749.583,A -85,B 0,C 180,E1 16748.21,E2 16748.21} C_VEL
LIN {X 0,Y 340.675,Z 758.574,A -85,B 0,C 180,E1 16744.885,E2 16744.885} C_VEL
LIN {X 0,Y 338.794,Z 766.255,A -85,B 0,C 180,E1 16741.355,E2 16741.355} C_VEL
LIN {X 0,Y 337.554,Z 772.306,A -85,B 0,C 180,E1 16737.796,E2 16737.796} C_VEL
LIN {X 0,Y 336.834,Z 776.664,A -85,B 0,C 180,E1 16734.21,E2 16734.21} C_VEL
LIN {X 0,Y 336.46,Z 779.52,A -85,B 0,C 180,E1 16730.596,E2 16730.596} C_VEL
LIN {X 0,Y 336.33,Z 780.894,A -85,B 0,C 180,E1 16727.12,E2 16727.12} C_VEL
LIN {X 0,Y 336.297,Z 780.766,A -85,B 0,C 180,E1 16723.774,E2 16723.774} C_VEL
LIN {X 0,Y 336.345,Z 779.26,A -85,B 0,C 180,E1 16720.194,E2 16720.194} C_VEL
LIN {X 0,Y 336.524,Z 776.533,A -85,B 0,C 180,E1 16716.912,E2 16716.912} C_VEL
LIN {X 0,Y 337.03,Z 771.917,A -85,B 0,C 180,E1 16713.251,E2 16713.251} C_VEL
LIN {X 0,Y 337.949,Z 765.97,A -85,B 0,C 180,E1 16709.761,E2 16709.761} C_VEL
LIN {X 0,Y 339.366,Z 758.484,A -85,B 0,C 180,E1 16706.369,E2 16706.369} C_VEL
LIN {X 0,Y 341.468,Z 748.994,A -85,B 0,C 180,E1 16702.905,E2 16702.905} C_VEL
LIN {X 0,Y 344.229,Z 737.797,A -85,B 0,C 180,E1 16699.555,E2 16699.555} C_VEL
LIN {X 0,Y 347.458,Z 725.449,A -85,B 0,C 180,E1 16696.484,E2 16696.484} C_VEL
LIN {X 0,Y 351.046,Z 711.82,A -85,B 0,C 180,E1 16693.665,E2 16693.665} C_VEL
LIN {X 0,Y 355.249,Z 695.838,A -85,B 0,C 180,E1 16690.883,E2 16690.883} C_VEL
LIN {X 0,Y 359.474,Z 679.237,A -85,B 0,C 180,E1 16688.455,E2 16688.455} C_VEL
LIN {X 0,Y 363.912,Z 660.89,A -85,B 0,C 180,E1 16686.209,E2 16686.209} C_VEL
LIN {X 0,Y 368.004,Z 642.265,A -85,B 0,C 180,E1 16684.32,E2 16684.32} C_VEL
LIN {X 0,Y 371.947,Z 622.442,A -85,B 0,C 180,E1 16682.644,E2 16682.644} C_VEL
LIN {X 0,Y 375.563,Z 601.927,A -85,B 0,C 180,E1 16681.225,E2 16681.225} C_VEL
LIN {X 0,Y 378.629,Z 581.228,A -85,B 0,C 180,E1 16680.082,E2 16680.082} C_VEL
LIN {X 0,Y 381.171,Z 559.687,A -85,B 0,C 180,E1 16679.161,E2 16679.161} C_VEL
LIN {X 0,Y 383.195,Z 536.883,A -85,B 0,C 180,E1 16678.451,E2 16678.451} C_VEL
LIN {X 0,Y 394.583,Z 350.069,A -85,B 0,C 180,E1 16674.357,E2 16674.357} C_VEL
LIN {X 0,Y 381.186,Z 329.996,A -85,B 0,C 180,E1 16671.505,E2 16671.505} C_VEL
LIN {X 0,Y 369.536,Z 313.411,A -85,B 0,C 180,E1 16668.784,E2 16668.784} C_VEL
LIN {X 0,Y 358.612,Z 298.534,A -85,B 0,C 180,E1 16665.983,E2 16665.983} C_VEL
LIN {X 0,Y 354.156,Z 292.782,A -85,B 0,C 180,E1 16664.763,E2 16664.763} C_VEL
LIN {X 0,Y 350.318,Z 287.671,A -85,B 0,C 180,E1 16663.663,E2 16663.663} C_VEL
LIN {X 0,Y 347.125,Z 283.497,A -85,B 0,C 180,E1 16662.731,E2 16662.731} C_VEL
LIN {X 0,Y 345.997,Z 282.1,A -85,B 0,C 180,E1 16662.396,E2 16662.396} C_VEL
LIN {X 0,Y 343.185,Z 278.682,A -85,B 0,C 180,E1 16661.535,E2 16661.535} C_VEL
LIN {X 0,Y 342.264,Z 276.756,A -85,B 0,C 180,E1 16661.203,E2 16661.203} C_VEL
LIN {X 0,Y 339.427,Z 274.344,A -85,B 0,C 180,E1 16660.353,E2 16660.353} C_VEL
LIN {X 0,Y 338.056,Z 271.249,A -85,B 0,C 180,E1 16659.836,E2 16659.836} C_VEL
LIN {X 0,Y 337.958,Z 270.639,A -85,B 0,C 180,E1 16659.753,E2 16659.753} C_VEL
LIN {X 0,Y 337.956,Z 270.626,A -85,B 0,C 180,E1 16655.604,E2 16655.604} C_VEL
LIN {X 0,Y 337.962,Z 270.628,A -85,B 0,C 180,E1 16651.358,E2 16651.358} C_VEL
LIN {X 0,Y 337.967,Z 270.633,A -85,B 0,C 180,E1 16647.119,E2 16647.119} C_VEL
LIN {X 0,Y 337.998,Z 270.62,A -85,B 0,C 180,E1 16642.694,E2 16642.694} C_VEL
LIN {X 0,Y 337.966,Z 270.622,A -85,B 0,C 180,E1 16638.289,E2 16638.289} C_VEL
LIN {X 0,Y 337.956,Z 270.625,A -85,B 0,C 180,E1 16634.031,E2 16634.031} C_VEL
LIN {X 0,Y 337.961,Z 270.637,A -85,B 0,C 180,E1 16632.087,E2 16632.087} C_VEL
LIN {X 0,Y 336.954,Z 270.757,A -85,B 0,C 180,E1 16630.781,E2 16630.781} C_VEL
LIN {X 0,Y 332.247,Z 271.352,A -85,B 0,C 180,E1 16628.218,E2 16628.218} C_VEL
LIN {X 0,Y 330.137,Z 271.601,A -85,B 0,C 180,E1 16626.51,E2 16626.51} C_VEL
LIN {X 0,Y 330.025,Z 271.613,A -85,B 0,C 180,E1 16626.121,E2 16626.121} C_VEL
LIN {X 0,Y 330.01,Z 271.615,A -85,B 0,C 180,E1 16621.796,E2 16621.796} C_VEL
LIN {X 0,Y 330.002,Z 271.617,A -85,B 0,C 180,E1 16617.571,E2 16617.571} C_VEL
LIN {X 0,Y 329.999,Z 271.618,A -85,B 0,C 180,E1 16613.139,E2 16613.139} C_VEL
LIN {X 0,Y 330.002,Z 271.621,A -85,B 0,C 180,E1 16608.895,E2 16608.895} C_VEL
LIN {X 0,Y 330.011,Z 271.622,A -85,B 0,C 180,E1 16604.606,E2 16604.606} C_VEL
LIN {X 0,Y 330.036,Z 271.618,A -85,B 0,C 180,E1 16600.183,E2 16600.183} C_VEL
LIN {X 0,Y 330.018,Z 271.62,A -85,B 0,C 180,E1 16595.78,E2 16595.78} C_VEL
LIN {X 0,Y 330.001,Z 271.624,A -85,B 0,C 180,E1 16591.405,E2 16591.405} C_VEL
LIN {X 0,Y 329.994,Z 271.627,A -85,B 0,C 180,E1 16587.224,E2 16587.224} C_VEL
LIN {X 0,Y 329.985,Z 271.629,A -85,B 0,C 180,E1 16582.817,E2 16582.817} C_VEL
LIN {X 0,Y 329.988,Z 271.626,A -85,B 0,C 180,E1 16578.496,E2 16578.496} C_VEL
LIN {X 0,Y 329.995,Z 271.621,A -85,B 0,C 180,E1 16574.204,E2 16574.204} C_VEL
LIN {X 0,Y 330.002,Z 271.621,A -85,B 0,C 180,E1 16569.942,E2 16569.942} C_VEL
LIN {X 0,Y 330.012,Z 271.628,A -85,B 0,C 180,E1 16565.736,E2 16565.736} C_VEL
LIN {X 0,Y 330.011,Z 271.624,A -85,B 0,C 180,E1 16561.387,E2 16561.387} C_VEL
LIN {X 0,Y 330.004,Z 271.622,A -85,B 0,C 180,E1 16557.219,E2 16557.219} C_VEL
LIN {X 0,Y 329.992,Z 271.631,A -85,B 0,C 180,E1 16552.862,E2 16552.862} C_VEL
LIN {X 0,Y 329.989,Z 271.623,A -85,B 0,C 180,E1 16548.639,E2 16548.639} C_VEL
LIN {X 0,Y 329.986,Z 271.627,A -85,B 0,C 180,E1 16544.353,E2 16544.353} C_VEL
LIN {X 0,Y 330.028,Z 271.669,A -85,B 0,C 180,E1 16541.358,E2 16541.358} C_VEL
LIN {X 0,Y 331.403,Z 275.261,A -85,B 0,C 180,E1 16540.267,E2 16540.267} C_VEL
LIN {X 0,Y 332.773,Z 276.798,A -85,B 0,C 180,E1 16539.6,E2 16539.6} C_VEL
LIN {X 0,Y 334.504,Z 280.625,A -85,B 0,C 180,E1 16538.427,E2 16538.427} C_VEL
LIN {X 0,Y 335.694,Z 282.513,A -85,B 0,C 180,E1 16537.772,E2 16537.772} C_VEL
LIN {X 0,Y 337.501,Z 285.749,A -85,B 0,C 180,E1 16536.84,E2 16536.84} C_VEL
LIN {X 0,Y 343.306,Z 293.767,A -85,B 0,C 180,E1 16534.926,E2 16534.926} C_VEL
LIN {X 0,Y 353.568,Z 308.153,A -85,B 0,C 180,E1 16531.817,E2 16531.817} C_VEL
LIN {X 0,Y 366.112,Z 326.821,A -85,B 0,C 180,E1 16528.374,E2 16528.374} C_VEL
LIN {X 0,Y 378.813,Z 346.888,A -85,B 0,C 180,E1 16525.217,E2 16525.217} C_VEL
LIN {X 0,Y 390.755,Z 367.125,A -85,B 0,C 180,E1 16522.503,E2 16522.503} C_VEL
LIN {X 0,Y 377.944,Z 565.902,A -85,B 0,C 180,E1 16518.082,E2 16518.082} C_VEL
LIN {X 0,Y 375.444,Z 602.488,A -85,B 0,C 180,E1 16517.197,E2 16517.197} C_VEL
LIN {X 0,Y 372.774,Z 625.213,A -85,B 0,C 180,E1 16516.434,E2 16516.434} C_VEL
LIN {X 0,Y 369.335,Z 647.785,A -85,B 0,C 180,E1 16515.394,E2 16515.394} C_VEL
LIN {X 0,Y 365.602,Z 668.711,A -85,B 0,C 180,E1 16514.138,E2 16514.138} C_VEL
LIN {X 0,Y 361.371,Z 689.638,A -85,B 0,C 180,E1 16512.578,E2 16512.578} C_VEL
LIN {X 0,Y 357.075,Z 708.926,A -85,B 0,C 180,E1 16510.828,E2 16510.828} C_VEL
LIN {X 0,Y 352.486,Z 727.936,A -85,B 0,C 180,E1 16508.732,E2 16508.732} C_VEL
LIN {X 0,Y 348.004,Z 745.658,A -85,B 0,C 180,E1 16506.394,E2 16506.394} C_VEL
LIN {X 0,Y 343.645,Z 762.483,A -85,B 0,C 180,E1 16503.758,E2 16503.758} C_VEL
LIN {X 0,Y 339.817,Z 777.446,A -85,B 0,C 180,E1 16500.989,E2 16500.989} C_VEL
LIN {X 0,Y 336.422,Z 790.944,A -85,B 0,C 180,E1 16498.005,E2 16498.005} C_VEL
LIN {X 0,Y 333.432,Z 803.784,A -85,B 0,C 180,E1 16494.632,E2 16494.632} C_VEL
LIN {X 0,Y 331.234,Z 814.522,A -85,B 0,C 180,E1 16491.235,E2 16491.235} C_VEL
LIN {X 0,Y 329.7,Z 823.471,A -85,B 0,C 180,E1 16487.775,E2 16487.775} C_VEL
LIN {X 0,Y 328.762,Z 830.726,A -85,B 0,C 180,E1 16484.259,E2 16484.259} C_VEL
LIN {X 0,Y 328.327,Z 836.43,A -85,B 0,C 180,E1 16480.704,E2 16480.704} C_VEL
LIN {X 0,Y 328.226,Z 840.194,A -85,B 0,C 180,E1 16477.349,E2 16477.349} C_VEL
LIN {X 0,Y 328.27,Z 842.633,A -85,B 0,C 180,E1 16473.84,E2 16473.84} C_VEL
LIN {X 0,Y 328.323,Z 843.404,A -85,B 0,C 180,E1 16470.696,E2 16470.696} C_VEL
LIN {X 0,Y 328.316,Z 842.84,A -85,B 0,C 180,E1 16467.328,E2 16467.328} C_VEL
LIN {X 0,Y 328.277,Z 840.77,A -85,B 0,C 180,E1 16464.054,E2 16464.054} C_VEL
LIN {X 0,Y 328.314,Z 837.051,A -85,B 0,C 180,E1 16460.533,E2 16460.533} C_VEL
LIN {X 0,Y 328.579,Z 831.901,A -85,B 0,C 180,E1 16457.164,E2 16457.164} C_VEL
LIN {X 0,Y 329.321,Z 824.348,A -85,B 0,C 180,E1 16453.416,E2 16453.416} C_VEL
LIN {X 0,Y 330.543,Z 815.777,A -85,B 0,C 180,E1 16450.011,E2 16450.011} C_VEL
LIN {X 0,Y 332.449,Z 804.997,A -85,B 0,C 180,E1 16446.538,E2 16446.538} C_VEL
LIN {X 0,Y 335.168,Z 791.896,A -85,B 0,C 180,E1 16443.034,E2 16443.034} C_VEL
LIN {X 0,Y 338.243,Z 778.495,A -85,B 0,C 180,E1 16440.013,E2 16440.013} C_VEL
LIN {X 0,Y 341.865,Z 763.443,A -85,B 0,C 180,E1 16437.142,E2 16437.142} C_VEL
LIN {X 0,Y 346.048,Z 746.548,A -85,B 0,C 180,E1 16434.401,E2 16434.401} C_VEL
LIN {X 0,Y 350.564,Z 728.603,A -85,B 0,C 180,E1 16431.926,E2 16431.926} C_VEL
LIN {X 0,Y 355.529,Z 708.528,A -85,B 0,C 180,E1 16429.59,E2 16429.59} C_VEL
LIN {X 0,Y 360.76,Z 686.945,A -85,B 0,C 180,E1 16427.497,E2 16427.497} C_VEL
LIN {X 0,Y 366.165,Z 663.869,A -85,B 0,C 180,E1 16425.649,E2 16425.649} C_VEL
LIN {X 0,Y 371.61,Z 639.591,A -85,B 0,C 180,E1 16424.077,E2 16424.077} C_VEL
LIN {X 0,Y 376.858,Z 614.734,A -85,B 0,C 180,E1 16422.81,E2 16422.81} C_VEL
LIN {X 0,Y 381.912,Z 587.833,A -85,B 0,C 180,E1 16421.742,E2 16421.742} C_VEL
LIN {X 0,Y 395.587,Z 500.979,A -85,B 0,C 180,E1 16419.079,E2 16419.079} C_VEL
LIN {X 0,Y 408.426,Z 435.976,A -85,B 0,C 180,E1 16417.132,E2 16417.132} C_VEL
LIN {X 0,Y 410.076,Z 428.427,A -85,B 0,C 180,E1 16416.896,E2 16416.896} C_VEL
LIN {X 0,Y 397.12,Z 490.659,A -85,B 0,C 180,E1 16415.051,E2 16415.051} C_VEL
LIN {X 0,Y 387.525,Z 546.888,A -85,B 0,C 180,E1 16413.339,E2 16413.339} C_VEL
LIN {X 0,Y 383.723,Z 571.028,A -85,B 0,C 180,E1 16412.432,E2 16412.432} C_VEL
LIN {X 0,Y 379.208,Z 595.211,A -85,B 0,C 180,E1 16411.207,E2 16411.207} C_VEL
LIN {X 0,Y 374.71,Z 616.141,A -85,B 0,C 180,E1 16409.855,E2 16409.855} C_VEL
LIN {X 0,Y 369.848,Z 636.6,A -85,B 0,C 180,E1 16408.237,E2 16408.237} C_VEL
LIN {X 0,Y 364.774,Z 656.206,A -85,B 0,C 180,E1 16406.364,E2 16406.364} C_VEL
LIN {X 0,Y 359.547,Z 674.923,A -85,B 0,C 180,E1 16404.209,E2 16404.209} C_VEL
LIN {X 0,Y 354.486,Z 691.983,A -85,B 0,C 180,E1 16401.86,E2 16401.86} C_VEL
LIN {X 0,Y 349.463,Z 708.067,A -85,B 0,C 180,E1 16399.212,E2 16399.212} C_VEL
LIN {X 0,Y 344.539,Z 723.289,A -85,B 0,C 180,E1 16396.178,E2 16396.178} C_VEL
LIN {X 0,Y 340.336,Z 736.155,A -85,B 0,C 180,E1 16393.076,E2 16393.076} C_VEL
LIN {X 0,Y 336.685,Z 747.573,A -85,B 0,C 180,E1 16389.748,E2 16389.748} C_VEL
LIN {X 0,Y 333.827,Z 757.127,A -85,B 0,C 180,E1 16386.365,E2 16386.365} C_VEL
LIN {X 0,Y 331.504,Z 765.652,A -85,B 0,C 180,E1 16382.595,E2 16382.595} C_VEL
LIN {X 0,Y 329.979,Z 771.927,A -85,B 0,C 180,E1 16378.961,E2 16378.961} C_VEL
LIN {X 0,Y 329.071,Z 776.656,A -85,B 0,C 180,E1 16375.288,E2 16375.288} C_VEL
LIN {X 0,Y 328.613,Z 779.771,A -85,B 0,C 180,E1 16371.781,E2 16371.781} C_VEL
LIN {X 0,Y 328.391,Z 781.39,A -85,B 0,C 180,E1 16368.232,E2 16368.232} C_VEL
LIN {X 0,Y 328.334,Z 781.697,A -85,B 0,C 180,E1 16364.64,E2 16364.64} C_VEL
LIN {X 0,Y 328.354,Z 780.627,A -85,B 0,C 180,E1 16361.268,E2 16361.268} C_VEL
LIN {X 0,Y 328.512,Z 778.066,A -85,B 0,C 180,E1 16357.642,E2 16357.642} C_VEL
LIN {X 0,Y 328.942,Z 774.078,A -85,B 0,C 180,E1 16354.046,E2 16354.046} C_VEL
LIN {X 0,Y 329.792,Z 768.298,A -85,B 0,C 180,E1 16350.388,E2 16350.388} C_VEL
LIN {X 0,Y 331.259,Z 760.698,A -85,B 0,C 180,E1 16346.682,E2 16346.682} C_VEL
LIN {X 0,Y 333.351,Z 751.599,A -85,B 0,C 180,E1 16343.142,E2 16343.142} C_VEL
LIN {X 0,Y 336.037,Z 740.99,A -85,B 0,C 180,E1 16339.788,E2 16339.788} C_VEL
LIN {X 0,Y 339.336,Z 728.64,A -85,B 0,C 180,E1 16336.569,E2 16336.569} C_VEL
LIN {X 0,Y 343.352,Z 714.088,A -85,B 0,C 180,E1 16333.414,E2 16333.414} C_VEL
LIN {X 0,Y 347.501,Z 699.019,A -85,B 0,C 180,E1 16330.678,E2 16330.678} C_VEL
LIN {X 0,Y 351.843,Z 682.737,A -85,B 0,C 180,E1 16328.194,E2 16328.194} C_VEL
LIN {X 0,Y 356.071,Z 665.873,A -85,B 0,C 180,E1 16326.035,E2 16326.035} C_VEL
LIN {X 0,Y 360.539,Z 646.863,A -85,B 0,C 180,E1 16323.99,E2 16323.99} C_VEL
LIN {X 0,Y 364.639,Z 627.699,A -85,B 0,C 180,E1 16322.27,E2 16322.27} C_VEL
LIN {X 0,Y 368.478,Z 606.924,A -85,B 0,C 180,E1 16320.759,E2 16320.759} C_VEL
LIN {X 0,Y 371.763,Z 586.063,A -85,B 0,C 180,E1 16319.538,E2 16319.538} C_VEL
LIN {X 0,Y 374.673,Z 563.562,A -85,B 0,C 180,E1 16318.514,E2 16318.514} C_VEL
LIN {X 0,Y 376.87,Z 541.443,A -85,B 0,C 180,E1 16317.771,E2 16317.771} C_VEL
LIN {X 0,Y 388.801,Z 353.757,A -85,B 0,C 180,E1 16313.581,E2 16313.581} C_VEL
LIN {X 0,Y 375.402,Z 333.503,A -85,B 0,C 180,E1 16310.626,E2 16310.626} C_VEL
LIN {X 0,Y 362.704,Z 315.447,A -85,B 0,C 180,E1 16307.532,E2 16307.532} C_VEL
LIN {X 0,Y 351.217,Z 299.948,A -85,B 0,C 180,E1 16304.426,E2 16304.426} C_VEL
LIN {X 0,Y 346.399,Z 293.848,A -85,B 0,C 180,E1 16303.055,E2 16303.055} C_VEL
LIN {X 0,Y 342.655,Z 288.863,A -85,B 0,C 180,E1 16301.916,E2 16301.916} C_VEL
LIN {X 0,Y 339.508,Z 284.73,A -85,B 0,C 180,E1 16300.909,E2 16300.909} C_VEL
LIN {X 0,Y 338.402,Z 283.329,A -85,B 0,C 180,E1 16300.557,E2 16300.557} C_VEL
LIN {X 0,Y 335.524,Z 280.064,A -85,B 0,C 180,E1 16299.636,E2 16299.636} C_VEL
LIN {X 0,Y 334.182,Z 277.671,A -85,B 0,C 180,E1 16299.148,E2 16299.148} C_VEL
LIN {X 0,Y 331.346,Z 275.134,A -85,B 0,C 180,E1 16298.232,E2 16298.232} C_VEL
LIN {X 0,Y 330.09,Z 272.086,A -85,B 0,C 180,E1 16297.704,E2 16297.704} C_VEL
LIN {X 0,Y 330.019,Z 271.619,A -85,B 0,C 180,E1 16297.619,E2 16297.619} C_VEL
LIN {X 0,Y 330.025,Z 271.619,A -85,B 0,C 180,E1 16293.302,E2 16293.302} C_VEL
LIN {X 0,Y 330.042,Z 271.608,A -85,B 0,C 180,E1 16288.96,E2 16288.96} C_VEL
LIN {X 0,Y 330.039,Z 271.612,A -85,B 0,C 180,E1 16284.613,E2 16284.613} C_VEL
LIN {X 0,Y 330.034,Z 271.621,A -85,B 0,C 180,E1 16280.41,E2 16280.41} C_VEL
LIN {X 0,Y 330.023,Z 271.625,A -85,B 0,C 180,E1 16276.154,E2 16276.154} C_VEL
LIN {X 0,Y 330.011,Z 271.626,A -85,B 0,C 180,E1 16271.818,E2 16271.818} C_VEL
LIN {X 0,Y 330.005,Z 271.626,A -85,B 0,C 180,E1 16267.372,E2 16267.372} C_VEL
LIN {X 0,Y 330.025,Z 271.613,A -85,B 0,C 180,E1 16266.121,E2 16266.121} C_VEL
LIN {X 0,Y 329.002,Z 271.749,A -85,B 0,C 180,E1 16264.784,E2 16264.784} C_VEL
LIN {X 0,Y 323.972,Z 272.375,A -85,B 0,C 180,E1 16261.967,E2 16261.967} C_VEL
LIN {X 0,Y 322.151,Z 272.604,A -85,B 0,C 180,E1 16260.308,E2 16260.308} C_VEL
LIN {X 0,Y 322.083,Z 272.617,A -85,B 0,C 180,E1 16260.009,E2 16260.009} C_VEL
LIN {X 0,Y 322.066,Z 272.622,A -85,B 0,C 180,E1 16255.599,E2 16255.599} C_VEL
LIN {X 0,Y 322.059,Z 272.622,A -85,B 0,C 180,E1 16251.165,E2 16251.165} C_VEL
LIN {X 0,Y 322.064,Z 272.62,A -85,B 0,C 180,E1 16246.845,E2 16246.845} C_VEL
LIN {X 0,Y 322.084,Z 272.616,A -85,B 0,C 180,E1 16242.371,E2 16242.371} C_VEL
LIN {X 0,Y 322.092,Z 272.612,A -85,B 0,C 180,E1 16237.96,E2 16237.96} C_VEL
LIN {X 0,Y 322.068,Z 272.612,A -85,B 0,C 180,E1 16233.542,E2 16233.542} C_VEL
LIN {X 0,Y 322.054,Z 272.611,A -85,B 0,C 180,E1 16229.168,E2 16229.168} C_VEL
LIN {X 0,Y 322.05,Z 272.609,A -85,B 0,C 180,E1 16224.776,E2 16224.776} C_VEL
LIN {X 0,Y 322.051,Z 272.614,A -85,B 0,C 180,E1 16220.535,E2 16220.535} C_VEL
LIN {X 0,Y 322.059,Z 272.617,A -85,B 0,C 180,E1 16216.222,E2 16216.222} C_VEL
LIN {X 0,Y 322.071,Z 272.616,A -85,B 0,C 180,E1 16211.821,E2 16211.821} C_VEL
LIN {X 0,Y 322.077,Z 272.609,A -85,B 0,C 180,E1 16207.489,E2 16207.489} C_VEL
LIN {X 0,Y 322.058,Z 272.613,A -85,B 0,C 180,E1 16203.201,E2 16203.201} C_VEL
LIN {X 0,Y 322.05,Z 272.621,A -85,B 0,C 180,E1 16198.93,E2 16198.93} C_VEL
LIN {X 0,Y 322.044,Z 272.612,A -85,B 0,C 180,E1 16194.475,E2 16194.475} C_VEL
LIN {X 0,Y 322.047,Z 272.621,A -85,B 0,C 180,E1 16190.166,E2 16190.166} C_VEL
LIN {X 0,Y 322.059,Z 272.611,A -85,B 0,C 180,E1 16185.801,E2 16185.801} C_VEL
LIN {X 0,Y 322.103,Z 272.806,A -85,B 0,C 180,E1 16183.497,E2 16183.497} C_VEL
LIN {X 0,Y 323.467,Z 276.264,A -85,B 0,C 180,E1 16182.365,E2 16182.365} C_VEL
LIN {X 0,Y 324.993,Z 278.231,A -85,B 0,C 180,E1 16181.523,E2 16181.523} C_VEL
LIN {X 0,Y 326.725,Z 281.798,A -85,B 0,C 180,E1 16180.327,E2 16180.327} C_VEL
LIN {X 0,Y 327.904,Z 283.74,A -85,B 0,C 180,E1 16179.628,E2 16179.628} C_VEL
LIN {X 0,Y 331.208,Z 288.121,A -85,B 0,C 180,E1 16178.434,E2 16178.434} C_VEL
LIN {X 0,Y 340.138,Z 300.653,A -85,B 0,C 180,E1 16175.373,E2 16175.373} C_VEL
LIN {X 0,Y 350.08,Z 314.745,A -85,B 0,C 180,E1 16172.299,E2 16172.299} C_VEL
LIN {X 0,Y 362.391,Z 333.249,A -85,B 0,C 180,E1 16168.845,E2 16168.845} C_VEL
LIN {X 0,Y 374.732,Z 352.965,A -85,B 0,C 180,E1 16165.713,E2 16165.713} C_VEL
LIN {X 0,Y 385.112,Z 370.695,A -85,B 0,C 180,E1 16163.3,E2 16163.3} C_VEL
LIN {X 0,Y 371.348,Z 574.933,A -85,B 0,C 180,E1 16158.681,E2 16158.681} C_VEL
LIN {X 0,Y 369.111,Z 604.273,A -85,B 0,C 180,E1 16157.934,E2 16157.934} C_VEL
LIN {X 0,Y 366.13,Z 627.641,A -85,B 0,C 180,E1 16157.106,E2 16157.106} C_VEL
LIN {X 0,Y 362.564,Z 649.959,A -85,B 0,C 180,E1 16156.033,E2 16156.033} C_VEL
LIN {X 0,Y 358.456,Z 671.873,A -85,B 0,C 180,E1 16154.658,E2 16154.658} C_VEL
LIN {X 0,Y 354.155,Z 691.874,A -85,B 0,C 180,E1 16153.093,E2 16153.093} C_VEL
LIN {X 0,Y 349.375,Z 712.146,A -85,B 0,C 180,E1 16151.162,E2 16151.162} C_VEL
LIN {X 0,Y 344.695,Z 730.873,A -85,B 0,C 180,E1 16149.007,E2 16149.007} C_VEL
LIN {X 0,Y 340.002,Z 748.666,A -85,B 0,C 180,E1 16146.552,E2 16146.552} C_VEL
LIN {X 0,Y 335.718,Z 764.442,A -85,B 0,C 180,E1 16143.944,E2 16143.944} C_VEL
LIN {X 0,Y 331.479,Z 780.227,A -85,B 0,C 180,E1 16140.847,E2 16140.847} C_VEL
LIN {X 0,Y 328.105,Z 793.359,A -85,B 0,C 180,E1 16137.789,E2 16137.789} C_VEL
LIN {X 0,Y 325.276,Z 805.101,A -85,B 0,C 180,E1 16134.51,E2 16134.51} C_VEL
LIN {X 0,Y 323.093,Z 815.463,A -85,B 0,C 180,E1 16131.035,E2 16131.035} C_VEL
LIN {X 0,Y 321.614,Z 824.05,A -85,B 0,C 180,E1 16127.549,E2 16127.549} C_VEL
LIN {X 0,Y 320.729,Z 830.819,A -85,B 0,C 180,E1 16124.071,E2 16124.071} C_VEL
LIN {X 0,Y 320.326,Z 836.265,A -85,B 0,C 180,E1 16120.428,E2 16120.428} C_VEL
LIN {X 0,Y 320.259,Z 839.889,A -85,B 0,C 180,E1 16116.992,E2 16116.992} C_VEL
LIN {X 0,Y 320.317,Z 842.056,A -85,B 0,C 180,E1 16113.398,E2 16113.398} C_VEL
LIN {X 0,Y 320.367,Z 842.665,A -85,B 0,C 180,E1 16110.177,E2 16110.177} C_VEL
LIN {X 0,Y 320.349,Z 841.831,A -85,B 0,C 180,E1 16106.778,E2 16106.778} C_VEL
LIN {X 0,Y 320.296,Z 839.703,A -85,B 0,C 180,E1 16103.546,E2 16103.546} C_VEL
LIN {X 0,Y 320.354,Z 835.761,A -85,B 0,C 180,E1 16099.932,E2 16099.932} C_VEL
LIN {X 0,Y 320.674,Z 830.462,A -85,B 0,C 180,E1 16096.475,E2 16096.475} C_VEL
LIN {X 0,Y 321.494,Z 823.081,A -85,B 0,C 180,E1 16092.814,E2 16092.814} C_VEL
LIN {X 0,Y 322.94,Z 813.856,A -85,B 0,C 180,E1 16089.14,E2 16089.14} C_VEL
LIN {X 0,Y 325.012,Z 803.115,A -85,B 0,C 180,E1 16085.653,E2 16085.653} C_VEL
LIN {X 0,Y 327.714,Z 790.978,A -85,B 0,C 180,E1 16082.369,E2 16082.369} C_VEL
LIN {X 0,Y 331.2,Z 776.822,A -85,B 0,C 180,E1 16079.12,E2 16079.12} C_VEL
LIN {X 0,Y 335.236,Z 761.16,A -85,B 0,C 180,E1 16076.099,E2 16076.099} C_VEL
LIN {X 0,Y 339.769,Z 744.069,A -85,B 0,C 180,E1 16073.316,E2 16073.316} C_VEL
LIN {X 0,Y 344.847,Z 725.072,A -85,B 0,C 180,E1 16070.699,E2 16070.699} C_VEL
LIN {X 0,Y 349.974,Z 705.952,A -85,B 0,C 180,E1 16068.464,E2 16068.464} C_VEL
LIN {X 0,Y 356.08,Z 682.567,A -85,B 0,C 180,E1 16066.192,E2 16066.192} C_VEL
LIN {X 0,Y 362.044,Z 659.021,A -85,B 0,C 180,E1 16064.332,E2 16064.332} C_VEL
LIN {X 0,Y 367.916,Z 635.078,A -85,B 0,C 180,E1 16062.796,E2 16062.796} C_VEL
LIN {X 0,Y 373.893,Z 609.444,A -85,B 0,C 180,E1 16061.515,E2 16061.515} C_VEL
LIN {X 0,Y 379.519,Z 582.089,A -85,B 0,C 180,E1 16060.441,E2 16060.441} C_VEL
LIN {X 0,Y 394.137,Z 501.191,A -85,B 0,C 180,E1 16057.926,E2 16057.926} C_VEL
LIN {X 0,Y 401.27,Z 467.703,A -85,B 0,C 180,E1 16056.902,E2 16056.902} C_VEL
LIN {X 0,Y 389.081,Z 525.709,A -85,B 0,C 180,E1 16055.151,E2 16055.151} C_VEL
LIN {X 0,Y 382.415,Z 562.742,A -85,B 0,C 180,E1 16053.923,E2 16053.923} C_VEL
LIN {X 0,Y 377.949,Z 585.216,A -85,B 0,C 180,E1 16052.889,E2 16052.889} C_VEL
LIN {X 0,Y 372.984,Z 606.968,A -85,B 0,C 180,E1 16051.608,E2 16051.608} C_VEL
LIN {X 0,Y 367.602,Z 628.424,A -85,B 0,C 180,E1 16050.033,E2 16050.033} C_VEL
LIN {X 0,Y 361.977,Z 649.006,A -85,B 0,C 180,E1 16048.188,E2 16048.188} C_VEL
LIN {X 0,Y 356.425,Z 667.915,A -85,B 0,C 180,E1 16046.133,E2 16046.133} C_VEL
LIN {X 0,Y 350.858,Z 685.699,A -85,B 0,C 180,E1 16043.825,E2 16043.825} C_VEL
LIN {X 0,Y 345.686,Z 701.558,A -85,B 0,C 180,E1 16041.375,E2 16041.375} C_VEL
LIN {X 0,Y 340.659,Z 716.253,A -85,B 0,C 180,E1 16038.66,E2 16038.66} C_VEL
LIN {X 0,Y 335.994,Z 729.595,A -85,B 0,C 180,E1 16035.714,E2 16035.714} C_VEL
LIN {X 0,Y 331.626,Z 742.206,A -85,B 0,C 180,E1 16032.363,E2 16032.363} C_VEL
LIN {X 0,Y 328.078,Z 752.793,A -85,B 0,C 180,E1 16028.944,E2 16028.944} C_VEL
LIN {X 0,Y 325.202,Z 761.946,A -85,B 0,C 180,E1 16025.295,E2 16025.295} C_VEL
LIN {X 0,Y 323.115,Z 769.201,A -85,B 0,C 180,E1 16021.598,E2 16021.598} C_VEL
LIN {X 0,Y 321.737,Z 774.863,A -85,B 0,C 180,E1 16017.865,E2 16017.865} C_VEL
LIN {X 0,Y 320.952,Z 778.984,A -85,B 0,C 180,E1 16014.102,E2 16014.102} C_VEL
LIN {X 0,Y 320.551,Z 781.399,A -85,B 0,C 180,E1 16010.487,E2 16010.487} C_VEL
LIN {X 0,Y 320.394,Z 782.496,A -85,B 0,C 180,E1 16006.651,E2 16006.651} C_VEL
LIN {X 0,Y 320.374,Z 782.189,A -85,B 0,C 180,E1 16003.317,E2 16003.317} C_VEL
LIN {X 0,Y 320.428,Z 780.5,A -85,B 0,C 180,E1 15999.738,E2 15999.738} C_VEL
LIN {X 0,Y 320.699,Z 777.435,A -85,B 0,C 180,E1 15996.093,E2 15996.093} C_VEL
LIN {X 0,Y 321.308,Z 772.654,A -85,B 0,C 180,E1 15992.38,E2 15992.38} C_VEL
LIN {X 0,Y 322.506,Z 765.934,A -85,B 0,C 180,E1 15988.495,E2 15988.495} C_VEL
LIN {X 0,Y 324.203,Z 758.249,A -85,B 0,C 180,E1 15985,E2 15985} C_VEL
LIN {X 0,Y 326.537,Z 748.853,A -85,B 0,C 180,E1 15981.572,E2 15981.572} C_VEL
LIN {X 0,Y 329.626,Z 737.454,A -85,B 0,C 180,E1 15978.143,E2 15978.143} C_VEL
LIN {X 0,Y 333.292,Z 724.608,A -85,B 0,C 180,E1 15974.933,E2 15974.933} C_VEL
LIN {X 0,Y 337.419,Z 710.329,A -85,B 0,C 180,E1 15971.951,E2 15971.951} C_VEL
LIN {X 0,Y 341.878,Z 694.485,A -85,B 0,C 180,E1 15969.198,E2 15969.198} C_VEL
LIN {X 0,Y 346.292,Z 678.193,A -85,B 0,C 180,E1 15966.819,E2 15966.819} C_VEL
LIN {X 0,Y 350.749,Z 660.896,A -85,B 0,C 180,E1 15964.683,E2 15964.683} C_VEL
LIN {X 0,Y 355.255,Z 641.65,A -85,B 0,C 180,E1 15962.704,E2 15962.704} C_VEL
LIN {X 0,Y 359.385,Z 621.968,A -85,B 0,C 180,E1 15961.037,E2 15961.037} C_VEL
LIN {X 0,Y 363.39,Z 600.205,A -85,B 0,C 180,E1 15959.538,E2 15959.538} C_VEL
LIN {X 0,Y 366.67,Z 578.975,A -85,B 0,C 180,E1 15958.374,E2 15958.374} C_VEL
LIN {X 0,Y 369.357,Z 556.895,A -85,B 0,C 180,E1 15957.449,E2 15957.449} C_VEL
LIN {X 0,Y 371.345,Z 534.531,A -85,B 0,C 180,E1 15956.782,E2 15956.782} C_VEL
LIN {X 0,Y 383.072,Z 357.368,A -85,B 0,C 180,E1 15952.786,E2 15952.786} C_VEL
LIN {X 0,Y 370.239,Z 338.027,A -85,B 0,C 180,E1 15949.874,E2 15949.874} C_VEL
LIN {X 0,Y 358.721,Z 321.556,A -85,B 0,C 180,E1 15946.991,E2 15946.991} C_VEL
LIN {X 0,Y 347.661,Z 306.505,A -85,B 0,C 180,E1 15943.939,E2 15943.939} C_VEL
LIN {X 0,Y 342.405,Z 299.8,A -85,B 0,C 180,E1 15942.395,E2 15942.395} C_VEL
LIN {X 0,Y 339.113,Z 295.354,A -85,B 0,C 180,E1 15941.352,E2 15941.352} C_VEL
LIN {X 0,Y 335.08,Z 290.123,A -85,B 0,C 180,E1 15940.057,E2 15940.057} C_VEL
LIN {X 0,Y 331.928,Z 286.224,A -85,B 0,C 180,E1 15939.013,E2 15939.013} C_VEL
LIN {X 0,Y 330.783,Z 284.536,A -85,B 0,C 180,E1 15938.607,E2 15938.607} C_VEL
LIN {X 0,Y 327.804,Z 281.318,A -85,B 0,C 180,E1 15937.59,E2 15937.59} C_VEL
LIN {X 0,Y 326.39,Z 278.734,A -85,B 0,C 180,E1 15937.035,E2 15937.035} C_VEL
LIN {X 0,Y 323.511,Z 276.274,A -85,B 0,C 180,E1 15936.034,E2 15936.034} C_VEL
LIN {X 0,Y 322.198,Z 273.287,A -85,B 0,C 180,E1 15935.455,E2 15935.455} C_VEL
LIN {X 0,Y 322.087,Z 272.602,A -85,B 0,C 180,E1 15935.345,E2 15935.345} C_VEL
LIN {X 0,Y 322.11,Z 272.607,A -85,B 0,C 180,E1 15930.891,E2 15930.891} C_VEL
LIN {X 0,Y 322.09,Z 272.6,A -85,B 0,C 180,E1 15926.442,E2 15926.442} C_VEL
LIN {X 0,Y 322.081,Z 272.599,A -85,B 0,C 180,E1 15922.151,E2 15922.151} C_VEL
LIN {X 0,Y 322.071,Z 272.602,A -85,B 0,C 180,E1 15917.815,E2 15917.815} C_VEL
LIN {X 0,Y 322.07,Z 272.608,A -85,B 0,C 180,E1 15913.407,E2 15913.407} C_VEL
LIN {X 0,Y 322.075,Z 272.61,A -85,B 0,C 180,E1 15909.086,E2 15909.086} C_VEL
LIN {X 0,Y 322.082,Z 272.61,A -85,B 0,C 180,E1 15904.833,E2 15904.833} C_VEL
LIN {X 0,Y 322.107,Z 272.609,A -85,B 0,C 180,E1 15900.353,E2 15900.353} C_VEL
LIN {X 0,Y 322.083,Z 272.617,A -85,B 0,C 180,E1 15900.009,E2 15900.009} C_VEL
LIN {X 0,Y 321.055,Z 272.759,A -85,B 0,C 180,E1 15898.639,E2 15898.639} C_VEL
LIN {X 0,Y 316.165,Z 273.363,A -85,B 0,C 180,E1 15895.85,E2 15895.85} C_VEL
LIN {X 0,Y 314.235,Z 273.59,A -85,B 0,C 180,E1 15894.152,E2 15894.152} C_VEL
LIN {X 0,Y 314.131,Z 273.598,A -85,B 0,C 180,E1 15893.744,E2 15893.744} C_VEL
LIN {X 0,Y 314.125,Z 273.603,A -85,B 0,C 180,E1 15889.512,E2 15889.512} C_VEL
LIN {X 0,Y 314.123,Z 273.604,A -85,B 0,C 180,E1 15884.956,E2 15884.956} C_VEL
LIN {X 0,Y 314.134,Z 273.602,A -85,B 0,C 180,E1 15880.477,E2 15880.477} C_VEL
LIN {X 0,Y 314.144,Z 273.6,A -85,B 0,C 180,E1 15876.061,E2 15876.061} C_VEL
LIN {X 0,Y 314.136,Z 273.602,A -85,B 0,C 180,E1 15871.676,E2 15871.676} C_VEL
LIN {X 0,Y 314.119,Z 273.605,A -85,B 0,C 180,E1 15867.278,E2 15867.278} C_VEL
LIN {X 0,Y 314.109,Z 273.607,A -85,B 0,C 180,E1 15862.848,E2 15862.848} C_VEL
LIN {X 0,Y 314.114,Z 273.601,A -85,B 0,C 180,E1 15858.365,E2 15858.365} C_VEL
LIN {X 0,Y 314.127,Z 273.597,A -85,B 0,C 180,E1 15853.996,E2 15853.996} C_VEL
LIN {X 0,Y 314.132,Z 273.602,A -85,B 0,C 180,E1 15849.524,E2 15849.524} C_VEL
LIN {X 0,Y 314.114,Z 273.609,A -85,B 0,C 180,E1 15845.111,E2 15845.111} C_VEL
LIN {X 0,Y 314.103,Z 273.601,A -85,B 0,C 180,E1 15840.727,E2 15840.727} C_VEL
LIN {X 0,Y 314.108,Z 273.609,A -85,B 0,C 180,E1 15836.165,E2 15836.165} C_VEL
LIN {X 0,Y 314.124,Z 273.6,A -85,B 0,C 180,E1 15831.763,E2 15831.763} C_VEL
LIN {X 0,Y 314.144,Z 273.604,A -85,B 0,C 180,E1 15827.311,E2 15827.311} C_VEL
LIN {X 0,Y 314.14,Z 273.763,A -85,B 0,C 180,E1 15825.858,E2 15825.858} C_VEL
LIN {X 0,Y 315.628,Z 277.386,A -85,B 0,C 180,E1 15824.566,E2 15824.566} C_VEL
LIN {X 0,Y 317.112,Z 279.245,A -85,B 0,C 180,E1 15823.701,E2 15823.701} C_VEL
LIN {X 0,Y 319.016,Z 282.999,A -85,B 0,C 180,E1 15822.393,E2 15822.393} C_VEL
LIN {X 0,Y 320.559,Z 284.923,A -85,B 0,C 180,E1 15821.776,E2 15821.776} C_VEL
LIN {X 0,Y 323.802,Z 289.218,A -85,B 0,C 180,E1 15820.517,E2 15820.517} C_VEL
LIN {X 0,Y 332.64,Z 301.465,A -85,B 0,C 180,E1 15817.277,E2 15817.277} C_VEL
LIN {X 0,Y 341.004,Z 313.22,A -85,B 0,C 180,E1 15814.512,E2 15814.512} C_VEL
LIN {X 0,Y 351.71,Z 328.913,A -85,B 0,C 180,E1 15811.284,E2 15811.284} C_VEL
LIN {X 0,Y 363.753,Z 347.768,A -85,B 0,C 180,E1 15807.982,E2 15807.982} C_VEL
LIN {X 0,Y 375.03,Z 366.418,A -85,B 0,C 180,E1 15805.164,E2 15805.164} C_VEL
LIN {X 0,Y 379.498,Z 374.393,A -85,B 0,C 180,E1 15804.113,E2 15804.113} C_VEL
LIN {X 0,Y 364.985,Z 580.862,A -85,B 0,C 180,E1 15799.373,E2 15799.373} C_VEL
LIN {X 0,Y 362.915,Z 605.263,A -85,B 0,C 180,E1 15798.717,E2 15798.717} C_VEL
LIN {X 0,Y 359.69,Z 629.081,A -85,B 0,C 180,E1 15797.842,E2 15797.842} C_VEL
LIN {X 0,Y 355.951,Z 651.319,A -85,B 0,C 180,E1 15796.732,E2 15796.732} C_VEL
LIN {X 0,Y 351.851,Z 672.371,A -85,B 0,C 180,E1 15795.383,E2 15795.383} C_VEL
LIN {X 0,Y 347.415,Z 692.144,A -85,B 0,C 180,E1 15793.798,E2 15793.798} C_VEL
LIN {X 0,Y 342.501,Z 712.164,A -85,B 0,C 180,E1 15791.851,E2 15791.851} C_VEL
LIN {X 0,Y 337.61,Z 730.932,A -85,B 0,C 180,E1 15789.643,E2 15789.643} C_VEL
LIN {X 0,Y 332.764,Z 748.633,A -85,B 0,C 180,E1 15787.15,E2 15787.15} C_VEL
LIN {X 0,Y 328.189,Z 764.816,A -85,B 0,C 180,E1 15784.41,E2 15784.41} C_VEL
LIN {X 0,Y 324.04,Z 779.664,A -85,B 0,C 180,E1 15781.428,E2 15781.428} C_VEL
LIN {X 0,Y 320.506,Z 792.819,A -85,B 0,C 180,E1 15778.304,E2 15778.304} C_VEL
LIN {X 0,Y 317.401,Z 805.159,A -85,B 0,C 180,E1 15774.767,E2 15774.767} C_VEL
LIN {X 0,Y 315.145,Z 815.395,A -85,B 0,C 180,E1 15771.202,E2 15771.202} C_VEL
LIN {X 0,Y 313.565,Z 824.223,A -85,B 0,C 180,E1 15767.44,E2 15767.44} C_VEL
LIN {X 0,Y 312.698,Z 830.867,A -85,B 0,C 180,E1 15763.873,E2 15763.873} C_VEL
LIN {X 0,Y 312.327,Z 836.072,A -85,B 0,C 180,E1 15760.139,E2 15760.139} C_VEL
LIN {X 0,Y 312.281,Z 839.548,A -85,B 0,C 180,E1 15756.617,E2 15756.617} C_VEL
LIN {X 0,Y 312.36,Z 841.401,A -85,B 0,C 180,E1 15753.118,E2 15753.118} C_VEL
LIN {X 0,Y 312.397,Z 841.899,A -85,B 0,C 180,E1 15749.631,E2 15749.631} C_VEL
LIN {X 0,Y 312.367,Z 840.786,A -85,B 0,C 180,E1 15746.144,E2 15746.144} C_VEL
LIN {X 0,Y 312.313,Z 838.313,A -85,B 0,C 180,E1 15742.641,E2 15742.641} C_VEL
LIN {X 0,Y 312.413,Z 834.223,A -85,B 0,C 180,E1 15739.114,E2 15739.114} C_VEL
LIN {X 0,Y 312.855,Z 828.327,A -85,B 0,C 180,E1 15735.374,E2 15735.374} C_VEL
LIN {X 0,Y 313.832,Z 820.772,A -85,B 0,C 180,E1 15731.702,E2 15731.702} C_VEL
LIN {X 0,Y 315.585,Z 810.874,A -85,B 0,C 180,E1 15727.849,E2 15727.849} C_VEL
LIN {X 0,Y 317.993,Z 799.749,A -85,B 0,C 180,E1 15724.282,E2 15724.282} C_VEL
LIN {X 0,Y 321.06,Z 787.214,A -85,B 0,C 180,E1 15720.932,E2 15720.932} C_VEL
LIN {X 0,Y 324.957,Z 772.524,A -85,B 0,C 180,E1 15717.629,E2 15717.629} C_VEL
LIN {X 0,Y 329.619,Z 755.917,A -85,B 0,C 180,E1 15714.485,E2 15714.485} C_VEL
LIN {X 0,Y 334.635,Z 738.418,A -85,B 0,C 180,E1 15711.683,E2 15711.683} C_VEL
LIN {X 0,Y 340.441,Z 718.184,A -85,B 0,C 180,E1 15708.972,E2 15708.972} C_VEL
LIN {X 0,Y 346.461,Z 697.099,A -85,B 0,C 180,E1 15706.617,E2 15706.617} C_VEL
LIN {X 0,Y 353.034,Z 673.842,A -85,B 0,C 180,E1 15704.461,E2 15704.461} C_VEL
LIN {X 0,Y 359.899,Z 649.007,A -85,B 0,C 180,E1 15702.589,E2 15702.589} C_VEL
LIN {X 0,Y 366.461,Z 624.846,A -85,B 0,C 180,E1 15701.144,E2 15701.144} C_VEL
LIN {X 0,Y 373.471,Z 596.997,A -85,B 0,C 180,E1 15699.852,E2 15699.852} C_VEL
LIN {X 0,Y 379.76,Z 568.487,A -85,B 0,C 180,E1 15698.822,E2 15698.822} C_VEL
LIN {X 0,Y 392.39,Z 507.016,A -85,B 0,C 180,E1 15696.91,E2 15696.91} C_VEL
LIN {X 0,Y 381.401,Z 558.514,A -85,B 0,C 180,E1 15695.28,E2 15695.28} C_VEL
LIN {X 0,Y 376.671,Z 580.296,A -85,B 0,C 180,E1 15694.339,E2 15694.339} C_VEL
LIN {X 0,Y 370.762,Z 603.688,A -85,B 0,C 180,E1 15693.009,E2 15693.009} C_VEL
LIN {X 0,Y 365.095,Z 624.352,A -85,B 0,C 180,E1 15691.541,E2 15691.541} C_VEL
LIN {X 0,Y 358.671,Z 645.864,A -85,B 0,C 180,E1 15689.659,E2 15689.659} C_VEL
LIN {X 0,Y 352.44,Z 665.688,A -85,B 0,C 180,E1 15687.545,E2 15687.545} C_VEL
LIN {X 0,Y 346.144,Z 684.456,A -85,B 0,C 180,E1 15685.128,E2 15685.128} C_VEL
LIN {X 0,Y 340.092,Z 701.582,A -85,B 0,C 180,E1 15682.472,E2 15682.472} C_VEL
LIN {X 0,Y 334.703,Z 716.274,A -85,B 0,C 180,E1 15679.73,E2 15679.73} C_VEL
LIN {X 0,Y 329.428,Z 730.389,A -85,B 0,C 180,E1 15676.579,E2 15676.579} C_VEL
LIN {X 0,Y 324.96,Z 742.392,A -85,B 0,C 180,E1 15673.344,E2 15673.344} C_VEL
LIN {X 0,Y 321.267,Z 752.58,A -85,B 0,C 180,E1 15670.039,E2 15670.039} C_VEL
LIN {X 0,Y 318.175,Z 761.432,A -85,B 0,C 180,E1 15666.498,E2 15666.498} C_VEL
LIN {X 0,Y 315.685,Z 769.317,A -85,B 0,C 180,E1 15662.544,E2 15662.544} C_VEL
LIN {X 0,Y 314.092,Z 775.163,A -85,B 0,C 180,E1 15658.726,E2 15658.726} C_VEL
LIN {X 0,Y 313.146,Z 779.397,A -85,B 0,C 180,E1 15654.873,E2 15654.873} C_VEL
LIN {X 0,Y 312.658,Z 781.977,A -85,B 0,C 180,E1 15651.173,E2 15651.173} C_VEL
LIN {X 0,Y 312.46,Z 783.264,A -85,B 0,C 180,E1 15647.423,E2 15647.423} C_VEL
LIN {X 0,Y 312.405,Z 783.04,A -85,B 0,C 180,E1 15643.775,E2 15643.775} C_VEL
LIN {X 0,Y 312.46,Z 781.444,A -85,B 0,C 180,E1 15639.98,E2 15639.98} C_VEL
LIN {X 0,Y 312.697,Z 778.604,A -85,B 0,C 180,E1 15636.444,E2 15636.444} C_VEL
LIN {X 0,Y 313.291,Z 774.041,A -85,B 0,C 180,E1 15632.644,E2 15632.644} C_VEL
LIN {X 0,Y 314.44,Z 767.772,A -85,B 0,C 180,E1 15628.785,E2 15628.785} C_VEL
LIN {X 0,Y 316.184,Z 760.001,A -85,B 0,C 180,E1 15625.088,E2 15625.088} C_VEL
LIN {X 0,Y 318.547,Z 750.818,A -85,B 0,C 180,E1 15621.58,E2 15621.58} C_VEL
LIN {X 0,Y 321.696,Z 739.694,A -85,B 0,C 180,E1 15618.073,E2 15618.073} C_VEL
LIN {X 0,Y 325.431,Z 727.126,A -85,B 0,C 180,E1 15614.792,E2 15614.792} C_VEL
LIN {X 0,Y 329.619,Z 712.992,A -85,B 0,C 180,E1 15611.742,E2 15611.742} C_VEL
LIN {X 0,Y 334.192,Z 697.431,A -85,B 0,C 180,E1 15608.926,E2 15608.926} C_VEL
LIN {X 0,Y 338.969,Z 680.565,A -85,B 0,C 180,E1 15606.364,E2 15606.364} C_VEL
LIN {X 0,Y 343.876,Z 662.269,A -85,B 0,C 180,E1 15604.044,E2 15604.044} C_VEL
LIN {X 0,Y 348.603,Z 642.768,A -85,B 0,C 180,E1 15602.004,E2 15602.004} C_VEL
LIN {X 0,Y 352.957,Z 622.798,A -85,B 0,C 180,E1 15600.282,E2 15600.282} C_VEL
LIN {X 0,Y 357.047,Z 601.383,A -85,B 0,C 180,E1 15598.783,E2 15598.783} C_VEL
LIN {X 0,Y 360.48,Z 580.046,A -85,B 0,C 180,E1 15597.591,E2 15597.591} C_VEL
LIN {X 0,Y 363.284,Z 557.853,A -85,B 0,C 180,E1 15596.646,E2 15596.646} C_VEL
LIN {X 0,Y 365.388,Z 535.208,A -85,B 0,C 180,E1 15595.957,E2 15595.957} C_VEL
LIN {X 0,Y 377.464,Z 361.133,A -85,B 0,C 180,E1 15591.969,E2 15591.969} C_VEL
LIN {X 0,Y 364.6,Z 341.683,A -85,B 0,C 180,E1 15588.95,E2 15588.95} C_VEL
LIN {X 0,Y 353.765,Z 326.305,A -85,B 0,C 180,E1 15586.166,E2 15586.166} C_VEL
LIN {X 0,Y 344.126,Z 313.05,A -85,B 0,C 180,E1 15583.442,E2 15583.442} C_VEL
LIN {X 0,Y 335.634,Z 301.904,A -85,B 0,C 180,E1 15580.819,E2 15580.819} C_VEL
LIN {X 0,Y 331.728,Z 296.841,A -85,B 0,C 180,E1 15579.544,E2 15579.544} C_VEL
LIN {X 0,Y 328.324,Z 292.309,A -85,B 0,C 180,E1 15578.363,E2 15578.363} C_VEL
LIN {X 0,Y 324.314,Z 287.531,A -85,B 0,C 180,E1 15576.947,E2 15576.947} C_VEL
LIN {X 0,Y 323.083,Z 285.679,A -85,B 0,C 180,E1 15576.479,E2 15576.479} C_VEL
LIN {X 0,Y 320.057,Z 282.534,A -85,B 0,C 180,E1 15575.379,E2 15575.379} C_VEL
LIN {X 0,Y 318.656,Z 279.822,A -85,B 0,C 180,E1 15574.771,E2 15574.771} C_VEL
LIN {X 0,Y 315.71,Z 277.457,A -85,B 0,C 180,E1 15573.679,E2 15573.679} C_VEL
LIN {X 0,Y 314.31,Z 274.436,A -85,B 0,C 180,E1 15573.011,E2 15573.011} C_VEL
LIN {X 0,Y 314.161,Z 273.589,A -85,B 0,C 180,E1 15572.875,E2 15572.875} C_VEL
LIN {X 0,Y 314.158,Z 273.587,A -85,B 0,C 180,E1 15568.543,E2 15568.543} C_VEL
LIN {X 0,Y 314.142,Z 273.597,A -85,B 0,C 180,E1 15564.156,E2 15564.156} C_VEL
LIN {X 0,Y 314.132,Z 273.601,A -85,B 0,C 180,E1 15559.735,E2 15559.735} C_VEL
LIN {X 0,Y 314.136,Z 273.596,A -85,B 0,C 180,E1 15555.25,E2 15555.25} C_VEL
LIN {X 0,Y 314.147,Z 273.592,A -85,B 0,C 180,E1 15550.865,E2 15550.865} C_VEL
LIN {X 0,Y 314.162,Z 273.589,A -85,B 0,C 180,E1 15546.424,E2 15546.424} C_VEL
LIN {X 0,Y 314.138,Z 273.592,A -85,B 0,C 180,E1 15541.899,E2 15541.899} C_VEL
LIN {X 0,Y 314.124,Z 273.594,A -85,B 0,C 180,E1 15537.504,E2 15537.504} C_VEL
LIN {X 0,Y 314.131,Z 273.598,A -85,B 0,C 180,E1 15533.744,E2 15533.744} C_VEL
LIN {X 0,Y 313.116,Z 273.726,A -85,B 0,C 180,E1 15532.339,E2 15532.339} C_VEL
LIN {X 0,Y 308.538,Z 274.304,A -85,B 0,C 180,E1 15529.68,E2 15529.68} C_VEL
LIN {X 0,Y 306.329,Z 274.57,A -85,B 0,C 180,E1 15527.841,E2 15527.841} C_VEL
LIN {X 0,Y 306.182,Z 274.593,A -85,B 0,C 180,E1 15527.317,E2 15527.317} C_VEL
LIN {X 0,Y 306.188,Z 274.593,A -85,B 0,C 180,E1 15522.718,E2 15522.718} C_VEL
LIN {X 0,Y 306.201,Z 274.587,A -85,B 0,C 180,E1 15518.343,E2 15518.343} C_VEL
LIN {X 0,Y 306.206,Z 274.583,A -85,B 0,C 180,E1 15513.939,E2 15513.939} C_VEL
LIN {X 0,Y 306.192,Z 274.582,A -85,B 0,C 180,E1 15509.54,E2 15509.54} C_VEL
LIN {X 0,Y 306.174,Z 274.583,A -85,B 0,C 180,E1 15505.118,E2 15505.118} C_VEL
LIN {X 0,Y 306.172,Z 274.59,A -85,B 0,C 180,E1 15500.649,E2 15500.649} C_VEL
LIN {X 0,Y 306.187,Z 274.595,A -85,B 0,C 180,E1 15496.112,E2 15496.112} C_VEL
LIN {X 0,Y 306.193,Z 274.591,A -85,B 0,C 180,E1 15491.596,E2 15491.596} C_VEL
LIN {X 0,Y 306.174,Z 274.589,A -85,B 0,C 180,E1 15487.126,E2 15487.126} C_VEL
LIN {X 0,Y 306.162,Z 274.598,A -85,B 0,C 180,E1 15482.618,E2 15482.618} C_VEL
LIN {X 0,Y 306.17,Z 274.593,A -85,B 0,C 180,E1 15478.126,E2 15478.126} C_VEL
LIN {X 0,Y 306.196,Z 274.59,A -85,B 0,C 180,E1 15473.623,E2 15473.623} C_VEL
LIN {X 0,Y 306.189,Z 274.588,A -85,B 0,C 180,E1 15469.08,E2 15469.08} C_VEL
LIN {X 0,Y 306.187,Z 274.723,A -85,B 0,C 180,E1 15468.409,E2 15468.409} C_VEL
LIN {X 0,Y 307.398,Z 277.909,A -85,B 0,C 180,E1 15467.219,E2 15467.219} C_VEL
LIN {X 0,Y 309.138,Z 279.951,A -85,B 0,C 180,E1 15466.15,E2 15466.15} C_VEL
LIN {X 0,Y 310.525,Z 282.84,A -85,B 0,C 180,E1 15465.261,E2 15465.261} C_VEL
LIN {X 0,Y 313.464,Z 286.404,A -85,B 0,C 180,E1 15463.982,E2 15463.982} C_VEL
LIN {X 0,Y 317.792,Z 292.242,A -85,B 0,C 180,E1 15462.181,E2 15462.181} C_VEL
LIN {X 0,Y 322.044,Z 297.985,A -85,B 0,C 180,E1 15460.501,E2 15460.501} C_VEL
LIN {X 0,Y 329.722,Z 308.647,A -85,B 0,C 180,E1 15457.676,E2 15457.676} C_VEL
LIN {X 0,Y 338.976,Z 321.748,A -85,B 0,C 180,E1 15454.583,E2 15454.583} C_VEL
LIN {X 0,Y 351.264,Z 340.221,A -85,B 0,C 180,E1 15450.871,E2 15450.871} C_VEL
LIN {X 0,Y 363.373,Z 359.685,A -85,B 0,C 180,E1 15447.572,E2 15447.572} C_VEL
LIN {X 0,Y 373.897,Z 377.607,A -85,B 0,C 180,E1 15444.954,E2 15444.954} C_VEL
LIN {X 0,Y 359.018,Z 580.663,A -85,B 0,C 180,E1 15440.221,E2 15440.221} C_VEL
LIN {X 0,Y 356.833,Z 605.224,A -85,B 0,C 180,E1 15439.547,E2 15439.547} C_VEL
LIN {X 0,Y 353.505,Z 628.897,A -85,B 0,C 180,E1 15438.661,E2 15438.661} C_VEL
LIN {X 0,Y 349.642,Z 651.057,A -85,B 0,C 180,E1 15437.541,E2 15437.541} C_VEL
LIN {X 0,Y 345.291,Z 672.621,A -85,B 0,C 180,E1 15436.136,E2 15436.136} C_VEL
LIN {X 0,Y 340.503,Z 693.243,A -85,B 0,C 180,E1 15434.451,E2 15434.451} C_VEL
LIN {X 0,Y 335.423,Z 713.102,A -85,B 0,C 180,E1 15432.464,E2 15432.464} C_VEL
LIN {X 0,Y 330.245,Z 732.126,A -85,B 0,C 180,E1 15430.154,E2 15430.154} C_VEL
LIN {X 0,Y 325.407,Z 749.087,A -85,B 0,C 180,E1 15427.692,E2 15427.692} C_VEL
LIN {X 0,Y 320.544,Z 765.653,A -85,B 0,C 180,E1 15424.805,E2 15424.805} C_VEL
LIN {X 0,Y 316.238,Z 780.381,A -85,B 0,C 180,E1 15421.731,E2 15421.731} C_VEL
LIN {X 0,Y 312.354,Z 794.239,A -85,B 0,C 180,E1 15418.276,E2 15418.276} C_VEL
LIN {X 0,Y 309.382,Z 805.756,A -85,B 0,C 180,E1 15414.841,E2 15414.841} C_VEL
LIN {X 0,Y 307.098,Z 815.806,A -85,B 0,C 180,E1 15411.184,E2 15411.184} C_VEL
LIN {X 0,Y 305.514,Z 824.397,A -85,B 0,C 180,E1 15407.324,E2 15407.324} C_VEL
LIN {X 0,Y 304.643,Z 831.153,A -85,B 0,C 180,E1 15403.473,E2 15403.473} C_VEL
LIN {X 0,Y 304.332,Z 835.869,A -85,B 0,C 180,E1 15399.835,E2 15399.835} C_VEL
LIN {X 0,Y 304.318,Z 839.212,A -85,B 0,C 180,E1 15396.033,E2 15396.033} C_VEL
LIN {X 0,Y 304.402,Z 840.732,A -85,B 0,C 180,E1 15392.822,E2 15392.822} C_VEL
LIN {X 0,Y 304.436,Z 841.059,A -85,B 0,C 180,E1 15389.245,E2 15389.245} C_VEL
LIN {X 0,Y 304.394,Z 839.921,A -85,B 0,C 180,E1 15385.854,E2 15385.854} C_VEL
LIN {X 0,Y 304.335,Z 837.358,A -85,B 0,C 180,E1 15382.257,E2 15382.257} C_VEL
LIN {X 0,Y 304.453,Z 833.168,A -85,B 0,C 180,E1 15378.634,E2 15378.634} C_VEL
LIN {X 0,Y 304.965,Z 827.183,A -85,B 0,C 180,E1 15374.792,E2 15374.792} C_VEL
LIN {X 0,Y 306.026,Z 819.764,A -85,B 0,C 180,E1 15371.126,E2 15371.126} C_VEL
LIN {X 0,Y 307.886,Z 810.062,A -85,B 0,C 180,E1 15367.264,E2 15367.264} C_VEL
LIN {X 0,Y 310.486,Z 798.988,A -85,B 0,C 180,E1 15363.613,E2 15363.613} C_VEL
LIN {X 0,Y 313.978,Z 785.734,A -85,B 0,C 180,E1 15360.001,E2 15360.001} C_VEL
LIN {X 0,Y 318.179,Z 770.999,A -85,B 0,C 180,E1 15356.636,E2 15356.636} C_VEL
LIN {X 0,Y 323.323,Z 753.875,A -85,B 0,C 180,E1 15353.354,E2 15353.354} C_VEL
LIN {X 0,Y 328.929,Z 735.811,A -85,B 0,C 180,E1 15350.443,E2 15350.443} C_VEL
LIN {X 0,Y 335.378,Z 715.035,A -85,B 0,C 180,E1 15347.64,E2 15347.64} C_VEL
LIN {X 0,Y 342.306,Z 692.765,A -85,B 0,C 180,E1 15345.16,E2 15345.16} C_VEL
LIN {X 0,Y 349.735,Z 668.737,A -85,B 0,C 180,E1 15342.954,E2 15342.954} C_VEL
LIN {X 0,Y 357.217,Z 644.495,A -85,B 0,C 180,E1 15341.153,E2 15341.153} C_VEL
LIN {X 0,Y 364.647,Z 619.92,A -85,B 0,C 180,E1 15339.71,E2 15339.71} C_VEL
LIN {X 0,Y 372.329,Z 592.817,A -85,B 0,C 180,E1 15338.481,E2 15338.481} C_VEL
LIN {X 0,Y 379.69,Z 563.22,A -85,B 0,C 180,E1 15337.442,E2 15337.442} C_VEL
LIN {X 0,Y 383.425,Z 546.476,A -85,B 0,C 180,E1 15336.912,E2 15336.912} C_VEL
LIN {X 0,Y 377.649,Z 571.163,A -85,B 0,C 180,E1 15336,E2 15336} C_VEL
LIN {X 0,Y 371.912,Z 592.547,A -85,B 0,C 180,E1 15334.936,E2 15334.936} C_VEL
LIN {X 0,Y 365.107,Z 615.05,A -85,B 0,C 180,E1 15333.493,E2 15333.493} C_VEL
LIN {X 0,Y 357.888,Z 637.342,A -85,B 0,C 180,E1 15331.685,E2 15331.685} C_VEL
LIN {X 0,Y 351.105,Z 657.344,A -85,B 0,C 180,E1 15329.705,E2 15329.705} C_VEL
LIN {X 0,Y 344.048,Z 677.051,A -85,B 0,C 180,E1 15327.336,E2 15327.336} C_VEL
LIN {X 0,Y 337.303,Z 695.153,A -85,B 0,C 180,E1 15324.708,E2 15324.708} C_VEL
LIN {X 0,Y 330.895,Z 711.585,A -85,B 0,C 180,E1 15321.82,E2 15321.82} C_VEL
LIN {X 0,Y 325.246,Z 725.663,A -85,B 0,C 180,E1 15318.834,E2 15318.834} C_VEL
LIN {X 0,Y 320.349,Z 737.809,A -85,B 0,C 180,E1 15315.758,E2 15315.758} C_VEL
LIN {X 0,Y 315.993,Z 748.803,A -85,B 0,C 180,E1 15312.427,E2 15312.427} C_VEL
LIN {X 0,Y 312.097,Z 758.927,A -85,B 0,C 180,E1 15308.662,E2 15308.662} C_VEL
LIN {X 0,Y 309.125,Z 767.113,A -85,B 0,C 180,E1 15304.826,E2 15304.826} C_VEL
LIN {X 0,Y 306.943,Z 773.878,A -85,B 0,C 180,E1 15300.749,E2 15300.749} C_VEL
LIN {X 0,Y 305.635,Z 778.746,A -85,B 0,C 180,E1 15296.815,E2 15296.815} C_VEL
LIN {X 0,Y 304.916,Z 781.888,A -85,B 0,C 180,E1 15293.034,E2 15293.034} C_VEL
LIN {X 0,Y 304.558,Z 783.731,A -85,B 0,C 180,E1 15289.001,E2 15289.001} C_VEL
LIN {X 0,Y 304.462,Z 784.091,A -85,B 0,C 180,E1 15285.161,E2 15285.161} C_VEL
LIN {X 0,Y 304.456,Z 782.974,A -85,B 0,C 180,E1 15281.428,E2 15281.428} C_VEL
LIN {X 0,Y 304.642,Z 780.322,A -85,B 0,C 180,E1 15277.421,E2 15277.421} C_VEL
LIN {X 0,Y 305.163,Z 776.263,A -85,B 0,C 180,E1 15273.542,E2 15273.542} C_VEL
LIN {X 0,Y 306.112,Z 770.727,A -85,B 0,C 180,E1 15269.804,E2 15269.804} C_VEL
LIN {X 0,Y 307.82,Z 763.101,A -85,B 0,C 180,E1 15265.814,E2 15265.814} C_VEL
LIN {X 0,Y 310.118,Z 754.411,A -85,B 0,C 180,E1 15262.179,E2 15262.179} C_VEL
LIN {X 0,Y 313.124,Z 743.896,A -85,B 0,C 180,E1 15258.627,E2 15258.627} C_VEL
LIN {X 0,Y 316.774,Z 731.857,A -85,B 0,C 180,E1 15255.252,E2 15255.252} C_VEL
LIN {X 0,Y 321.071,Z 718.076,A -85,B 0,C 180,E1 15252.033,E2 15252.033} C_VEL
LIN {X 0,Y 325.78,Z 702.845,A -85,B 0,C 180,E1 15249.065,E2 15249.065} C_VEL
LIN {X 0,Y 330.58,Z 686.645,A -85,B 0,C 180,E1 15246.441,E2 15246.441} C_VEL
LIN {X 0,Y 335.497,Z 669.169,A -85,B 0,C 180,E1 15244.061,E2 15244.061} C_VEL
LIN {X 0,Y 340.198,Z 651.331,A -85,B 0,C 180,E1 15242.021,E2 15242.021} C_VEL
LIN {X 0,Y 344.891,Z 631.453,A -85,B 0,C 180,E1 15240.146,E2 15240.146} C_VEL
LIN {X 0,Y 349.114,Z 611.059,A -85,B 0,C 180,E1 15238.575,E2 15238.575} C_VEL
LIN {X 0,Y 353.009,Z 589.076,A -85,B 0,C 180,E1 15237.213,E2 15237.213} C_VEL
LIN {X 0,Y 356.218,Z 567.088,A -85,B 0,C 180,E1 15236.154,E2 15236.154} C_VEL
LIN {X 0,Y 358.722,Z 544.688,A -85,B 0,C 180,E1 15235.357,E2 15235.357} C_VEL
LIN {X 0,Y 362.337,Z 494.747,A -85,B 0,C 180,E1 15234.152,E2 15234.152} C_VEL
LIN {X 0,Y 371.764,Z 364.726,A -85,B 0,C 180,E1 15231.126,E2 15231.126} C_VEL
LIN {X 0,Y 359.214,Z 345.797,A -85,B 0,C 180,E1 15228.082,E2 15228.082} C_VEL
LIN {X 0,Y 347.738,Z 329.3,A -85,B 0,C 180,E1 15224.999,E2 15224.999} C_VEL
LIN {X 0,Y 336.763,Z 314.377,A -85,B 0,C 180,E1 15221.736,E2 15221.736} C_VEL
LIN {X 0,Y 328.415,Z 303.54,A -85,B 0,C 180,E1 15219.022,E2 15219.022} C_VEL
LIN {X 0,Y 324.074,Z 297.97,A -85,B 0,C 180,E1 15217.492,E2 15217.492} C_VEL
LIN {X 0,Y 320.724,Z 293.585,A -85,B 0,C 180,E1 15216.266,E2 15216.266} C_VEL
LIN {X 0,Y 316.743,Z 288.94,A -85,B 0,C 180,E1 15214.755,E2 15214.755} C_VEL
LIN {X 0,Y 315.371,Z 286.818,A -85,B 0,C 180,E1 15214.183,E2 15214.183} C_VEL
LIN {X 0,Y 312.362,Z 283.778,A -85,B 0,C 180,E1 15212.998,E2 15212.998} C_VEL
LIN {X 0,Y 310.882,Z 280.893,A -85,B 0,C 180,E1 15212.306,E2 15212.306} C_VEL
LIN {X 0,Y 307.927,Z 278.614,A -85,B 0,C 180,E1 15211.118,E2 15211.118} C_VEL
LIN {X 0,Y 306.377,Z 275.501,A -85,B 0,C 180,E1 15210.329,E2 15210.329} C_VEL
LIN {X 0,Y 306.201,Z 274.584,A -85,B 0,C 180,E1 15210.189,E2 15210.189} C_VEL
LIN {X 0,Y 306.193,Z 274.575,A -85,B 0,C 180,E1 15205.695,E2 15205.695} C_VEL
LIN {X 0,Y 306.199,Z 274.578,A -85,B 0,C 180,E1 15201.363,E2 15201.363} C_VEL
LIN {X 0,Y 306.221,Z 274.586,A -85,B 0,C 180,E1 15196.79,E2 15196.79} C_VEL
LIN {X 0,Y 306.217,Z 274.593,A -85,B 0,C 180,E1 15192.324,E2 15192.324} C_VEL
LIN {X 0,Y 306.198,Z 274.594,A -85,B 0,C 180,E1 15187.946,E2 15187.946} C_VEL
LIN {X 0,Y 306.19,Z 274.595,A -85,B 0,C 180,E1 15183.427,E2 15183.427} C_VEL
LIN {X 0,Y 306.196,Z 274.595,A -85,B 0,C 180,E1 15178.943,E2 15178.943} C_VEL
LIN {X 0,Y 306.213,Z 274.591,A -85,B 0,C 180,E1 15174.388,E2 15174.388} C_VEL
LIN {X 0,Y 306.21,Z 274.593,A -85,B 0,C 180,E1 15169.968,E2 15169.968} C_VEL
LIN {X 0,Y 306.182,Z 274.593,A -85,B 0,C 180,E1 15167.317,E2 15167.317} C_VEL
LIN {X 0,Y 305.176,Z 274.735,A -85,B 0,C 180,E1 15165.876,E2 15165.876} C_VEL
LIN {X 0,Y 300.742,Z 275.297,A -85,B 0,C 180,E1 15163.25,E2 15163.25} C_VEL
LIN {X 0,Y 298.434,Z 275.569,A -85,B 0,C 180,E1 15161.366,E2 15161.366} C_VEL
LIN {X 0,Y 298.247,Z 275.583,A -85,B 0,C 180,E1 15160.721,E2 15160.721} C_VEL
LIN {X 0,Y 298.264,Z 275.579,A -85,B 0,C 180,E1 15156.153,E2 15156.153} C_VEL
LIN {X 0,Y 298.251,Z 275.58,A -85,B 0,C 180,E1 15151.528,E2 15151.528} C_VEL
LIN {X 0,Y 298.237,Z 275.583,A -85,B 0,C 180,E1 15147.122,E2 15147.122} C_VEL
LIN {X 0,Y 298.238,Z 275.58,A -85,B 0,C 180,E1 15142.466,E2 15142.466} C_VEL
LIN {X 0,Y 298.255,Z 275.573,A -85,B 0,C 180,E1 15137.961,E2 15137.961} C_VEL
LIN {X 0,Y 298.259,Z 275.575,A -85,B 0,C 180,E1 15133.56,E2 15133.56} C_VEL
LIN {X 0,Y 298.235,Z 275.588,A -85,B 0,C 180,E1 15129.063,E2 15129.063} C_VEL
LIN {X 0,Y 298.224,Z 275.582,A -85,B 0,C 180,E1 15124.42,E2 15124.42} C_VEL
LIN {X 0,Y 298.246,Z 275.579,A -85,B 0,C 180,E1 15119.805,E2 15119.805} C_VEL
LIN {X 0,Y 298.249,Z 275.579,A -85,B 0,C 180,E1 15115.19,E2 15115.19} C_VEL
LIN {X 0,Y 298.273,Z 275.708,A -85,B 0,C 180,E1 15111.176,E2 15111.176} C_VEL
LIN {X 0,Y 299.326,Z 278.733,A -85,B 0,C 180,E1 15109.995,E2 15109.995} C_VEL
LIN {X 0,Y 301.713,Z 281.579,A -85,B 0,C 180,E1 15108.626,E2 15108.626} C_VEL
LIN {X 0,Y 304.606,Z 285.713,A -85,B 0,C 180,E1 15107.197,E2 15107.197} C_VEL
LIN {X 0,Y 306.415,Z 287.776,A -85,B 0,C 180,E1 15106.361,E2 15106.361} C_VEL
LIN {X 0,Y 309.632,Z 292.121,A -85,B 0,C 180,E1 15104.902,E2 15104.902} C_VEL
LIN {X 0,Y 314.904,Z 299.338,A -85,B 0,C 180,E1 15102.633,E2 15102.633} C_VEL
LIN {X 0,Y 319.237,Z 305.268,A -85,B 0,C 180,E1 15100.893,E2 15100.893} C_VEL
LIN {X 0,Y 326.563,Z 315.475,A -85,B 0,C 180,E1 15098.159,E2 15098.159} C_VEL
LIN {X 0,Y 335.719,Z 328.664,A -85,B 0,C 180,E1 15095.027,E2 15095.027} C_VEL
LIN {X 0,Y 347.379,Z 346.319,A -85,B 0,C 180,E1 15091.433,E2 15091.433} C_VEL
LIN {X 0,Y 359.331,Z 365.726,A -85,B 0,C 180,E1 15088.105,E2 15088.105} C_VEL
LIN {X 0,Y 368.383,Z 381.331,A -85,B 0,C 180,E1 15085.801,E2 15085.801} C_VEL
LIN {X 0,Y 351.711,Z 597.214,A -85,B 0,C 180,E1 15080.651,E2 15080.651} C_VEL
LIN {X 0,Y 348.671,Z 620.828,A -85,B 0,C 180,E1 15079.839,E2 15079.839} C_VEL
LIN {X 0,Y 344.982,Z 642.461,A -85,B 0,C 180,E1 15078.833,E2 15078.833} C_VEL
LIN {X 0,Y 340.5,Z 664.827,A -85,B 0,C 180,E1 15077.477,E2 15077.477} C_VEL
LIN {X 0,Y 335.674,Z 685.787,A -85,B 0,C 180,E1 15075.875,E2 15075.875} C_VEL
LIN {X 0,Y 330.488,Z 706.243,A -85,B 0,C 180,E1 15073.94,E2 15073.94} C_VEL
LIN {X 0,Y 325.174,Z 725.301,A -85,B 0,C 180,E1 15071.733,E2 15071.733} C_VEL
LIN {X 0,Y 319.957,Z 743.078,A -85,B 0,C 180,E1 15069.255,E2 15069.255} C_VEL
LIN {X 0,Y 314.856,Z 760.01,A -85,B 0,C 180,E1 15066.427,E2 15066.427} C_VEL
LIN {X 0,Y 310.256,Z 775.149,A -85,B 0,C 180,E1 15063.416,E2 15063.416} C_VEL
LIN {X 0,Y 306.004,Z 789.36,A -85,B 0,C 180,E1 15059.992,E2 15059.992} C_VEL
LIN {X 0,Y 302.605,Z 801.454,A -85,B 0,C 180,E1 15056.489,E2 15056.489} C_VEL
LIN {X 0,Y 299.92,Z 812.194,A -85,B 0,C 180,E1 15052.748,E2 15052.748} C_VEL
LIN {X 0,Y 298.039,Z 821.202,A -85,B 0,C 180,E1 15048.902,E2 15048.902} C_VEL
LIN {X 0,Y 296.92,Z 828.33,A -85,B 0,C 180,E1 15045.026,E2 15045.026} C_VEL
LIN {X 0,Y 296.409,Z 833.99,A -85,B 0,C 180,E1 15040.998,E2 15040.998} C_VEL
LIN {X 0,Y 296.33,Z 837.554,A -85,B 0,C 180,E1 15037.365,E2 15037.365} C_VEL
LIN {X 0,Y 296.413,Z 839.687,A -85,B 0,C 180,E1 15033.673,E2 15033.673} C_VEL
LIN {X 0,Y 296.477,Z 840.314,A -85,B 0,C 180,E1 15030.385,E2 15030.385} C_VEL
LIN {X 0,Y 296.442,Z 839.631,A -85,B 0,C 180,E1 15026.711,E2 15026.711} C_VEL
LIN {X 0,Y 296.38,Z 837.517,A -85,B 0,C 180,E1 15023.217,E2 15023.217} C_VEL
LIN {X 0,Y 296.422,Z 833.678,A -85,B 0,C 180,E1 15019.307,E2 15019.307} C_VEL
LIN {X 0,Y 296.82,Z 828.364,A -85,B 0,C 180,E1 15015.564,E2 15015.564} C_VEL
LIN {X 0,Y 297.835,Z 821.106,A -85,B 0,C 180,E1 15011.603,E2 15011.603} C_VEL
LIN {X 0,Y 299.686,Z 811.744,A -85,B 0,C 180,E1 15007.547,E2 15007.547} C_VEL
LIN {X 0,Y 302.378,Z 800.604,A -85,B 0,C 180,E1 15003.653,E2 15003.653} C_VEL
LIN {X 0,Y 306.095,Z 787.281,A -85,B 0,C 180,E1 14999.797,E2 14999.797} C_VEL
LIN {X 0,Y 310.428,Z 773.096,A -85,B 0,C 180,E1 14996.357,E2 14996.357} C_VEL
LIN {X 0,Y 315.948,Z 756.008,A -85,B 0,C 180,E1 14992.893,E2 14992.893} C_VEL
LIN {X 0,Y 321.684,Z 738.614,A -85,B 0,C 180,E1 14989.953,E2 14989.953} C_VEL
LIN {X 0,Y 328.794,Z 717.483,A -85,B 0,C 180,E1 14986.943,E2 14986.943} C_VEL
LIN {X 0,Y 336.56,Z 694.701,A -85,B 0,C 180,E1 14984.276,E2 14984.276} C_VEL
LIN {X 0,Y 345.141,Z 669.727,A -85,B 0,C 180,E1 14981.881,E2 14981.881} C_VEL
LIN {X 0,Y 353.345,Z 646.06,A -85,B 0,C 180,E1 14980.053,E2 14980.053} C_VEL
LIN {X 0,Y 361.487,Z 622.533,A -85,B 0,C 180,E1 14978.611,E2 14978.611} C_VEL
LIN {X 0,Y 370.377,Z 595.471,A -85,B 0,C 180,E1 14977.341,E2 14977.341} C_VEL
LIN {X 0,Y 374.605,Z 581.499,A -85,B 0,C 180,E1 14976.8,E2 14976.8} C_VEL
LIN {X 0,Y 367.253,Z 604.067,A -85,B 0,C 180,E1 14975.541,E2 14975.541} C_VEL
LIN {X 0,Y 359.84,Z 624.869,A -85,B 0,C 180,E1 14974.05,E2 14974.05} C_VEL
LIN {X 0,Y 352.001,Z 645.892,A -85,B 0,C 180,E1 14972.182,E2 14972.182} C_VEL
LIN {X 0,Y 344.413,Z 665.548,A -85,B 0,C 180,E1 14970.053,E2 14970.053} C_VEL
LIN {X 0,Y 336.685,Z 684.982,A -85,B 0,C 180,E1 14967.505,E2 14967.505} C_VEL
LIN {X 0,Y 329.913,Z 701.328,A -85,B 0,C 180,E1 14964.916,E2 14964.916} C_VEL
LIN {X 0,Y 322.988,Z 717.678,A -85,B 0,C 180,E1 14961.809,E2 14961.809} C_VEL
LIN {X 0,Y 316.645,Z 732.336,A -85,B 0,C 180,E1 14958.409,E2 14958.409} C_VEL
LIN {X 0,Y 311.265,Z 744.761,A -85,B 0,C 180,E1 14954.893,E2 14954.893} C_VEL
LIN {X 0,Y 306.62,Z 755.703,A -85,B 0,C 180,E1 14951.095,E2 14951.095} C_VEL
LIN {X 0,Y 302.839,Z 765.088,A -85,B 0,C 180,E1 14947.019,E2 14947.019} C_VEL
LIN {X 0,Y 300.078,Z 772.47,A -85,B 0,C 180,E1 14942.867,E2 14942.867} C_VEL
LIN {X 0,Y 298.31,Z 777.861,A -85,B 0,C 180,E1 14938.85,E2 14938.85} C_VEL
LIN {X 0,Y 297.248,Z 781.839,A -85,B 0,C 180,E1 14934.672,E2 14934.672} C_VEL
LIN {X 0,Y 296.724,Z 784.103,A -85,B 0,C 180,E1 14930.695,E2 14930.695} C_VEL
LIN {X 0,Y 296.515,Z 784.883,A -85,B 0,C 180,E1 14926.747,E2 14926.747} C_VEL
LIN {X 0,Y 296.485,Z 784.383,A -85,B 0,C 180,E1 14922.942,E2 14922.942} C_VEL
LIN {X 0,Y 296.568,Z 782.368,A -85,B 0,C 180,E1 14919.052,E2 14919.052} C_VEL
LIN {X 0,Y 296.971,Z 778.709,A -85,B 0,C 180,E1 14914.902,E2 14914.902} C_VEL
LIN {X 0,Y 297.829,Z 773.575,A -85,B 0,C 180,E1 14910.874,E2 14910.874} C_VEL
LIN {X 0,Y 299.266,Z 766.889,A -85,B 0,C 180,E1 14906.995,E2 14906.995} C_VEL
LIN {X 0,Y 301.491,Z 758.334,A -85,B 0,C 180,E1 14903.06,E2 14903.06} C_VEL
LIN {X 0,Y 304.431,Z 748.372,A -85,B 0,C 180,E1 14899.35,E2 14899.35} C_VEL
LIN {X 0,Y 308.12,Z 736.595,A -85,B 0,C 180,E1 14895.764,E2 14895.764} C_VEL
LIN {X 0,Y 312.271,Z 723.64,A -85,B 0,C 180,E1 14892.503,E2 14892.503} C_VEL
LIN {X 0,Y 317.132,Z 708.507,A -85,B 0,C 180,E1 14889.326,E2 14889.326} C_VEL
LIN {X 0,Y 322.016,Z 692.965,A -85,B 0,C 180,E1 14886.597,E2 14886.597} C_VEL
LIN {X 0,Y 327.122,Z 675.761,A -85,B 0,C 180,E1 14884.08,E2 14884.08} C_VEL
LIN {X 0,Y 332.064,Z 657.832,A -85,B 0,C 180,E1 14881.891,E2 14881.891} C_VEL
LIN {X 0,Y 337.135,Z 637.756,A -85,B 0,C 180,E1 14879.857,E2 14879.857} C_VEL
LIN {X 0,Y 341.698,Z 617.527,A -85,B 0,C 180,E1 14878.175,E2 14878.175} C_VEL
LIN {X 0,Y 345.706,Z 596.692,A -85,B 0,C 180,E1 14876.779,E2 14876.779} C_VEL
LIN {X 0,Y 349.179,Z 574.791,A -85,B 0,C 180,E1 14875.62,E2 14875.62} C_VEL
LIN {X 0,Y 352.123,Z 551.308,A -85,B 0,C 180,E1 14874.69,E2 14874.69} C_VEL
LIN {X 0,Y 354.28,Z 527.284,A -85,B 0,C 180,E1 14874.025,E2 14874.025} C_VEL
LIN {X 0,Y 366.202,Z 368.575,A -85,B 0,C 180,E1 14870.29,E2 14870.29} C_VEL
LIN {X 0,Y 354.654,Z 351.049,A -85,B 0,C 180,E1 14867.411,E2 14867.411} C_VEL
LIN {X 0,Y 343.678,Z 335.253,A -85,B 0,C 180,E1 14864.396,E2 14864.396} C_VEL
LIN {X 0,Y 333.33,Z 321.021,A -85,B 0,C 180,E1 14861.245,E2 14861.245} C_VEL
LIN {X 0,Y 325.009,Z 310.088,A -85,B 0,C 180,E1 14858.449,E2 14858.449} C_VEL
LIN {X 0,Y 320.738,Z 304.64,A -85,B 0,C 180,E1 14856.94,E2 14856.94} C_VEL
LIN {X 0,Y 316.65,Z 299.377,A -85,B 0,C 180,E1 14855.392,E2 14855.392} C_VEL
LIN {X 0,Y 313.339,Z 295.155,A -85,B 0,C 180,E1 14854.073,E2 14854.073} C_VEL
LIN {X 0,Y 312.11,Z 293.663,A -85,B 0,C 180,E1 14853.583,E2 14853.583} C_VEL
LIN {X 0,Y 309.049,Z 290.12,A -85,B 0,C 180,E1 14852.329,E2 14852.329} C_VEL
LIN {X 0,Y 307.853,Z 288.067,A -85,B 0,C 180,E1 14851.77,E2 14851.77} C_VEL
LIN {X 0,Y 304.824,Z 285.207,A -85,B 0,C 180,E1 14850.481,E2 14850.481} C_VEL
LIN {X 0,Y 302.946,Z 281.887,A -85,B 0,C 180,E1 14849.537,E2 14849.537} C_VEL
LIN {X 0,Y 299.794,Z 279.371,A -85,B 0,C 180,E1 14848.139,E2 14848.139} C_VEL
LIN {X 0,Y 298.433,Z 276.501,A -85,B 0,C 180,E1 14847.362,E2 14847.362} C_VEL
LIN {X 0,Y 298.27,Z 275.577,A -85,B 0,C 180,E1 14847.177,E2 14847.177} C_VEL
LIN {X 0,Y 298.3,Z 275.562,A -85,B 0,C 180,E1 14842.684,E2 14842.684} C_VEL
LIN {X 0,Y 298.26,Z 275.566,A -85,B 0,C 180,E1 14838.006,E2 14838.006} C_VEL
LIN {X 0,Y 298.254,Z 275.572,A -85,B 0,C 180,E1 14833.446,E2 14833.446} C_VEL
LIN {X 0,Y 298.264,Z 275.576,A -85,B 0,C 180,E1 14828.982,E2 14828.982} C_VEL
LIN {X 0,Y 298.274,Z 275.577,A -85,B 0,C 180,E1 14824.594,E2 14824.594} C_VEL
LIN {X 0,Y 298.268,Z 275.582,A -85,B 0,C 180,E1 14820.037,E2 14820.037} C_VEL
LIN {X 0,Y 298.247,Z 275.589,A -85,B 0,C 180,E1 14815.492,E2 14815.492} C_VEL
LIN {X 0,Y 298.25,Z 275.589,A -85,B 0,C 180,E1 14810.934,E2 14810.934} C_VEL
LIN {X 0,Y 298.267,Z 275.587,A -85,B 0,C 180,E1 14806.387,E2 14806.387} C_VEL
LIN {X 0,Y 298.265,Z 275.589,A -85,B 0,C 180,E1 14801.839,E2 14801.839} C_VEL
LIN {X 0,Y 298.247,Z 275.583,A -85,B 0,C 180,E1 14800.721,E2 14800.721} C_VEL
LIN {X 0,Y 297.407,Z 275.683,A -85,B 0,C 180,E1 14799.346,E2 14799.346} C_VEL
LIN {X 0,Y 293.762,Z 276.148,A -85,B 0,C 180,E1 14797.067,E2 14797.067} C_VEL
LIN {X 0,Y 290.672,Z 276.515,A -85,B 0,C 180,E1 14794.828,E2 14794.828} C_VEL
LIN {X 0,Y 290.324,Z 276.56,A -85,B 0,C 180,E1 14793.945,E2 14793.945} C_VEL
LIN {X 0,Y 290.303,Z 276.563,A -85,B 0,C 180,E1 14789.276,E2 14789.276} C_VEL
LIN {X 0,Y 290.299,Z 276.563,A -85,B 0,C 180,E1 14784.6,E2 14784.6} C_VEL
LIN {X 0,Y 290.311,Z 276.57,A -85,B 0,C 180,E1 14780.142,E2 14780.142} C_VEL
LIN {X 0,Y 290.32,Z 276.572,A -85,B 0,C 180,E1 14775.58,E2 14775.58} C_VEL
LIN {X 0,Y 290.29,Z 276.566,A -85,B 0,C 180,E1 14770.917,E2 14770.917} C_VEL
LIN {X 0,Y 290.29,Z 276.57,A -85,B 0,C 180,E1 14766.325,E2 14766.325} C_VEL
LIN {X 0,Y 290.309,Z 276.573,A -85,B 0,C 180,E1 14761.774,E2 14761.774} C_VEL
LIN {X 0,Y 290.308,Z 276.565,A -85,B 0,C 180,E1 14757.234,E2 14757.234} C_VEL
LIN {X 0,Y 290.302,Z 276.661,A -85,B 0,C 180,E1 14754.265,E2 14754.265} C_VEL
LIN {X 0,Y 291.349,Z 279.624,A -85,B 0,C 180,E1 14753.198,E2 14753.198} C_VEL
LIN {X 0,Y 293.576,Z 282.082,A -85,B 0,C 180,E1 14751.971,E2 14751.971} C_VEL
LIN {X 0,Y 294.636,Z 283.085,A -85,B 0,C 180,E1 14751.41,E2 14751.41} C_VEL
LIN {X 0,Y 297.197,Z 286.706,A -85,B 0,C 180,E1 14750.02,E2 14750.02} C_VEL
LIN {X 0,Y 299.102,Z 288.928,A -85,B 0,C 180,E1 14749.062,E2 14749.062} C_VEL
LIN {X 0,Y 302.464,Z 293.425,A -85,B 0,C 180,E1 14747.396,E2 14747.396} C_VEL
LIN {X 0,Y 304.235,Z 295.877,A -85,B 0,C 180,E1 14746.552,E2 14746.552} C_VEL
LIN {X 0,Y 308.27,Z 301.287,A -85,B 0,C 180,E1 14744.718,E2 14744.718} C_VEL
LIN {X 0,Y 311.998,Z 306.399,A -85,B 0,C 180,E1 14743.09,E2 14743.09} C_VEL
LIN {X 0,Y 316.652,Z 312.818,A -85,B 0,C 180,E1 14741.209,E2 14741.209} C_VEL
LIN {X 0,Y 324.058,Z 323.235,A -85,B 0,C 180,E1 14738.41,E2 14738.41} C_VEL
LIN {X 0,Y 332.92,Z 336.277,A -85,B 0,C 180,E1 14735.324,E2 14735.324} C_VEL
LIN {X 0,Y 343.385,Z 352.212,A -85,B 0,C 180,E1 14732.042,E2 14732.042} C_VEL
LIN {X 0,Y 355.132,Z 371.426,A -85,B 0,C 180,E1 14728.703,E2 14728.703} C_VEL
LIN {X 0,Y 362.854,Z 385.036,A -85,B 0,C 180,E1 14726.667,E2 14726.667} C_VEL
LIN {X 0,Y 345.859,Z 596.565,A -85,B 0,C 180,E1 14721.557,E2 14721.557} C_VEL
LIN {X 0,Y 342.716,Z 620.229,A -85,B 0,C 180,E1 14720.734,E2 14720.734} C_VEL
LIN {X 0,Y 338.995,Z 641.419,A -85,B 0,C 180,E1 14719.742,E2 14719.742} C_VEL
LIN {X 0,Y 334.372,Z 663.84,A -85,B 0,C 180,E1 14718.376,E2 14718.376} C_VEL
LIN {X 0,Y 329.385,Z 684.853,A -85,B 0,C 180,E1 14716.76,E2 14716.76} C_VEL
LIN {X 0,Y 324.043,Z 705.209,A -85,B 0,C 180,E1 14714.818,E2 14714.818} C_VEL
LIN {X 0,Y 318.502,Z 724.424,A -85,B 0,C 180,E1 14712.568,E2 14712.568} C_VEL
LIN {X 0,Y 313.079,Z 742.241,A -85,B 0,C 180,E1 14710.051,E2 14710.051} C_VEL
LIN {X 0,Y 307.766,Z 759.208,A -85,B 0,C 180,E1 14707.173,E2 14707.173} C_VEL
LIN {X 0,Y 302.875,Z 774.642,A -85,B 0,C 180,E1 14704.042,E2 14704.042} C_VEL
LIN {X 0,Y 298.496,Z 788.72,A -85,B 0,C 180,E1 14700.584,E2 14700.584} C_VEL
LIN {X 0,Y 294.953,Z 800.793,A -85,B 0,C 180,E1 14697.014,E2 14697.014} C_VEL
LIN {X 0,Y 292.126,Z 811.558,A -85,B 0,C 180,E1 14693.177,E2 14693.177} C_VEL
LIN {X 0,Y 290.143,Z 820.578,A -85,B 0,C 180,E1 14689.222,E2 14689.222} C_VEL
LIN {X 0,Y 288.966,Z 827.679,A -85,B 0,C 180,E1 14685.244,E2 14685.244} C_VEL
LIN {X 0,Y 288.438,Z 833.237,A -85,B 0,C 180,E1 14681.177,E2 14681.177} C_VEL
LIN {X 0,Y 288.357,Z 836.694,A -85,B 0,C 180,E1 14677.569,E2 14677.569} C_VEL
LIN {X 0,Y 288.446,Z 838.887,A -85,B 0,C 180,E1 14673.774,E2 14673.774} C_VEL
LIN {X 0,Y 288.516,Z 839.523,A -85,B 0,C 180,E1 14670.395,E2 14670.395} C_VEL
LIN {X 0,Y 288.477,Z 838.957,A -85,B 0,C 180,E1 14666.819,E2 14666.819} C_VEL
LIN {X 0,Y 288.396,Z 836.763,A -85,B 0,C 180,E1 14663.028,E2 14663.028} C_VEL
LIN {X 0,Y 288.437,Z 833.17,A -85,B 0,C 180,E1 14659.209,E2 14659.209} C_VEL
LIN {X 0,Y 288.887,Z 827.619,A -85,B 0,C 180,E1 14655.158,E2 14655.158} C_VEL
LIN {X 0,Y 290.077,Z 819.941,A -85,B 0,C 180,E1 14650.884,E2 14650.884} C_VEL
LIN {X 0,Y 292.074,Z 810.746,A -85,B 0,C 180,E1 14646.815,E2 14646.815} C_VEL
LIN {X 0,Y 294.88,Z 800.033,A -85,B 0,C 180,E1 14642.975,E2 14642.975} C_VEL
LIN {X 0,Y 298.672,Z 787.424,A -85,B 0,C 180,E1 14639.188,E2 14639.188} C_VEL
LIN {X 0,Y 303.243,Z 773.52,A -85,B 0,C 180,E1 14635.678,E2 14635.678} C_VEL
LIN {X 0,Y 309.1,Z 756.591,A -85,B 0,C 180,E1 14632.12,E2 14632.12} C_VEL
LIN {X 0,Y 315.597,Z 738.456,A -85,B 0,C 180,E1 14628.942,E2 14628.942} C_VEL
LIN {X 0,Y 323.348,Z 717.328,A -85,B 0,C 180,E1 14625.841,E2 14625.841} C_VEL
LIN {X 0,Y 332.222,Z 693.704,A -85,B 0,C 180,E1 14623,E2 14623} C_VEL
LIN {X 0,Y 341.995,Z 668.29,A -85,B 0,C 180,E1 14620.522,E2 14620.522} C_VEL
LIN {X 0,Y 351.105,Z 645.16,A -85,B 0,C 180,E1 14618.712,E2 14618.712} C_VEL
LIN {X 0,Y 360.157,Z 622.296,A -85,B 0,C 180,E1 14617.308,E2 14617.308} C_VEL
LIN {X 0,Y 365.516,Z 608.236,A -85,B 0,C 180,E1 14616.609,E2 14616.609} C_VEL
LIN {X 0,Y 356.876,Z 629.334,A -85,B 0,C 180,E1 14615.056,E2 14615.056} C_VEL
LIN {X 0,Y 347.59,Z 651.117,A -85,B 0,C 180,E1 14613.034,E2 14613.034} C_VEL
LIN {X 0,Y 338.526,Z 671.912,A -85,B 0,C 180,E1 14610.632,E2 14610.632} C_VEL
LIN {X 0,Y 330.217,Z 690.692,A -85,B 0,C 180,E1 14607.992,E2 14607.992} C_VEL
LIN {X 0,Y 322.567,Z 707.566,A -85,B 0,C 180,E1 14605.131,E2 14605.131} C_VEL
LIN {X 0,Y 315.091,Z 723.683,A -85,B 0,C 180,E1 14601.796,E2 14601.796} C_VEL
LIN {X 0,Y 308.865,Z 736.937,A -85,B 0,C 180,E1 14598.465,E2 14598.465} C_VEL
LIN {X 0,Y 303.387,Z 748.562,A -85,B 0,C 180,E1 14594.898,E2 14594.898} C_VEL
LIN {X 0,Y 298.833,Z 758.448,A -85,B 0,C 180,E1 14591.192,E2 14591.192} C_VEL
LIN {X 0,Y 295.253,Z 766.705,A -85,B 0,C 180,E1 14587.396,E2 14587.396} C_VEL
LIN {X 0,Y 292.342,Z 773.95,A -85,B 0,C 180,E1 14583.14,E2 14583.14} C_VEL
LIN {X 0,Y 290.391,Z 779.356,A -85,B 0,C 180,E1 14578.819,E2 14578.819} C_VEL
LIN {X 0,Y 289.272,Z 783.102,A -85,B 0,C 180,E1 14574.449,E2 14574.449} C_VEL
LIN {X 0,Y 288.755,Z 785.15,A -85,B 0,C 180,E1 14570.436,E2 14570.436} C_VEL
LIN {X 0,Y 288.554,Z 785.697,A -85,B 0,C 180,E1 14566.579,E2 14566.579} C_VEL
LIN {X 0,Y 288.517,Z 785.014,A -85,B 0,C 180,E1 14562.664,E2 14562.664} C_VEL
LIN {X 0,Y 288.613,Z 783.03,A -85,B 0,C 180,E1 14558.885,E2 14558.885} C_VEL
LIN {X 0,Y 289.053,Z 779.257,A -85,B 0,C 180,E1 14554.604,E2 14554.604} C_VEL
LIN {X 0,Y 289.923,Z 774.352,A -85,B 0,C 180,E1 14550.682,E2 14550.682} C_VEL
LIN {X 0,Y 291.427,Z 767.662,A -85,B 0,C 180,E1 14546.709,E2 14546.709} C_VEL
LIN {X 0,Y 293.736,Z 759.173,A -85,B 0,C 180,E1 14542.711,E2 14542.711} C_VEL
LIN {X 0,Y 296.781,Z 749.289,A -85,B 0,C 180,E1 14538.936,E2 14538.936} C_VEL
LIN {X 0,Y 300.454,Z 737.964,A -85,B 0,C 180,E1 14535.403,E2 14535.403} C_VEL
LIN {X 0,Y 304.831,Z 724.818,A -85,B 0,C 180,E1 14532.002,E2 14532.002} C_VEL
LIN {X 0,Y 309.864,Z 709.726,A -85,B 0,C 180,E1 14528.757,E2 14528.757} C_VEL
LIN {X 0,Y 314.95,Z 694.139,A -85,B 0,C 180,E1 14525.955,E2 14525.955} C_VEL
LIN {X 0,Y 320.298,Z 676.72,A -85,B 0,C 180,E1 14523.36,E2 14523.36} C_VEL
LIN {X 0,Y 325.609,Z 658.111,A -85,B 0,C 180,E1 14521.055,E2 14521.055} C_VEL
LIN {X 0,Y 330.961,Z 637.549,A -85,B 0,C 180,E1 14518.957,E2 14518.957} C_VEL
LIN {X 0,Y 335.693,Z 617.051,A -85,B 0,C 180,E1 14517.25,E2 14517.25} C_VEL
LIN {X 0,Y 339.954,Z 595.527,A -85,B 0,C 180,E1 14515.805,E2 14515.805} C_VEL
LIN {X 0,Y 343.625,Z 572.69,A -85,B 0,C 180,E1 14514.617,E2 14514.617} C_VEL
LIN {X 0,Y 346.464,Z 550.109,A -85,B 0,C 180,E1 14513.743,E2 14513.743} C_VEL
LIN {X 0,Y 349.127,Z 519.49,A -85,B 0,C 180,E1 14512.927,E2 14512.927} C_VEL
LIN {X 0,Y 360.675,Z 372.297,A -85,B 0,C 180,E1 14509.411,E2 14509.411} C_VEL
LIN {X 0,Y 347.576,Z 352.347,A -85,B 0,C 180,E1 14505.99,E2 14505.99} C_VEL
LIN {X 0,Y 336.012,Z 336.006,A -85,B 0,C 180,E1 14502.644,E2 14502.644} C_VEL
LIN {X 0,Y 326.074,Z 322.44,A -85,B 0,C 180,E1 14499.444,E2 14499.444} C_VEL
LIN {X 0,Y 317.673,Z 311.546,A -85,B 0,C 180,E1 14496.462,E2 14496.462} C_VEL
LIN {X 0,Y 313.522,Z 306.198,A -85,B 0,C 180,E1 14494.85,E2 14494.85} C_VEL
LIN {X 0,Y 309.98,Z 301.498,A -85,B 0,C 180,E1 14493.423,E2 14493.423} C_VEL
LIN {X 0,Y 306.153,Z 297.087,A -85,B 0,C 180,E1 14491.822,E2 14491.822} C_VEL
LIN {X 0,Y 304.854,Z 295.135,A -85,B 0,C 180,E1 14491.223,E2 14491.223} C_VEL
LIN {X 0,Y 301.657,Z 291.691,A -85,B 0,C 180,E1 14489.812,E2 14489.812} C_VEL
LIN {X 0,Y 300.127,Z 289.166,A -85,B 0,C 180,E1 14489.047,E2 14489.047} C_VEL
LIN {X 0,Y 296.91,Z 286.187,A -85,B 0,C 180,E1 14487.546,E2 14487.546} C_VEL
LIN {X 0,Y 295.318,Z 283,A -85,B 0,C 180,E1 14486.615,E2 14486.615} C_VEL
LIN {X 0,Y 292.262,Z 280.847,A -85,B 0,C 180,E1 14485.145,E2 14485.145} C_VEL
LIN {X 0,Y 290.587,Z 277.826,A -85,B 0,C 180,E1 14484.127,E2 14484.127} C_VEL
LIN {X 0,Y 290.318,Z 276.568,A -85,B 0,C 180,E1 14483.873,E2 14483.873} C_VEL
LIN {X 0,Y 290.321,Z 276.56,A -85,B 0,C 180,E1 14479.284,E2 14479.284} C_VEL
LIN {X 0,Y 290.347,Z 276.553,A -85,B 0,C 180,E1 14474.613,E2 14474.613} C_VEL
LIN {X 0,Y 290.325,Z 276.556,A -85,B 0,C 180,E1 14470.068,E2 14470.068} C_VEL
LIN {X 0,Y 290.312,Z 276.559,A -85,B 0,C 180,E1 14465.591,E2 14465.591} C_VEL
LIN {X 0,Y 290.318,Z 276.561,A -85,B 0,C 180,E1 14460.951,E2 14460.951} C_VEL
LIN {X 0,Y 290.334,Z 276.562,A -85,B 0,C 180,E1 14456.33,E2 14456.33} C_VEL
LIN {X 0,Y 290.313,Z 276.569,A -85,B 0,C 180,E1 14451.692,E2 14451.692} C_VEL
LIN {X 0,Y 290.305,Z 276.574,A -85,B 0,C 180,E1 14447.008,E2 14447.008} C_VEL
LIN {X 0,Y 290.322,Z 276.572,A -85,B 0,C 180,E1 14442.451,E2 14442.451} C_VEL
LIN {X 0,Y 290.333,Z 276.567,A -85,B 0,C 180,E1 14437.946,E2 14437.946} C_VEL
LIN {X 0,Y 290.324,Z 276.56,A -85,B 0,C 180,E1 14433.945,E2 14433.945} C_VEL
LIN {X 0,Y 289.463,Z 276.682,A -85,B 0,C 180,E1 14432.532,E2 14432.532} C_VEL
LIN {X 0,Y 285.809,Z 277.148,A -85,B 0,C 180,E1 14430.191,E2 14430.191} C_VEL
LIN {X 0,Y 282.714,Z 277.524,A -85,B 0,C 180,E1 14427.89,E2 14427.89} C_VEL
LIN {X 0,Y 282.358,Z 277.557,A -85,B 0,C 180,E1 14426.982,E2 14426.982} C_VEL
LIN {X 0,Y 282.37,Z 277.554,A -85,B 0,C 180,E1 14422.261,E2 14422.261} C_VEL
LIN {X 0,Y 282.379,Z 277.55,A -85,B 0,C 180,E1 14417.725,E2 14417.725} C_VEL
LIN {X 0,Y 282.357,Z 277.558,A -85,B 0,C 180,E1 14413.096,E2 14413.096} C_VEL
LIN {X 0,Y 282.352,Z 277.564,A -85,B 0,C 180,E1 14408.345,E2 14408.345} C_VEL
LIN {X 0,Y 282.369,Z 277.554,A -85,B 0,C 180,E1 14403.652,E2 14403.652} C_VEL
LIN {X 0,Y 282.359,Z 277.566,A -85,B 0,C 180,E1 14398.983,E2 14398.983} C_VEL
LIN {X 0,Y 282.384,Z 277.7,A -85,B 0,C 180,E1 14397.841,E2 14397.841} C_VEL
LIN {X 0,Y 283.434,Z 280.679,A -85,B 0,C 180,E1 14396.964,E2 14396.964} C_VEL
LIN {X 0,Y 285.986,Z 283.297,A -85,B 0,C 180,E1 14395.385,E2 14395.385} C_VEL
LIN {X 0,Y 287.574,Z 284.4,A -85,B 0,C 180,E1 14394.511,E2 14394.511} C_VEL
LIN {X 0,Y 290.034,Z 288.477,A -85,B 0,C 180,E1 14392.958,E2 14392.958} C_VEL
LIN {X 0,Y 292.14,Z 290.502,A -85,B 0,C 180,E1 14391.832,E2 14391.832} C_VEL
LIN {X 0,Y 295.038,Z 294.37,A -85,B 0,C 180,E1 14390.242,E2 14390.242} C_VEL
LIN {X 0,Y 296.751,Z 296.652,A -85,B 0,C 180,E1 14389.367,E2 14389.367} C_VEL
LIN {X 0,Y 301.125,Z 302.438,A -85,B 0,C 180,E1 14387.192,E2 14387.192} C_VEL
LIN {X 0,Y 308.547,Z 312.535,A -85,B 0,C 180,E1 14383.816,E2 14383.816} C_VEL
LIN {X 0,Y 316.69,Z 323.952,A -85,B 0,C 180,E1 14380.494,E2 14380.494} C_VEL
LIN {X 0,Y 326.215,Z 337.802,A -85,B 0,C 180,E1 14376.994,E2 14376.994} C_VEL
LIN {X 0,Y 336.815,Z 353.981,A -85,B 0,C 180,E1 14373.485,E2 14373.485} C_VEL
LIN {X 0,Y 347.969,Z 372.17,A -85,B 0,C 180,E1 14370.142,E2 14370.142} C_VEL
LIN {X 0,Y 357.393,Z 388.347,A -85,B 0,C 180,E1 14367.562,E2 14367.562} C_VEL
LIN {X 0,Y 339.981,Z 596.007,A -85,B 0,C 180,E1 14362.471,E2 14362.471} C_VEL
LIN {X 0,Y 336.721,Z 619.796,A -85,B 0,C 180,E1 14361.634,E2 14361.634} C_VEL
LIN {X 0,Y 332.818,Z 641.334,A -85,B 0,C 180,E1 14360.612,E2 14360.612} C_VEL
LIN {X 0,Y 328.053,Z 663.683,A -85,B 0,C 180,E1 14359.231,E2 14359.231} C_VEL
LIN {X 0,Y 322.918,Z 684.621,A -85,B 0,C 180,E1 14357.598,E2 14357.598} C_VEL
LIN {X 0,Y 317.372,Z 705.081,A -85,B 0,C 180,E1 14355.619,E2 14355.619} C_VEL
LIN {X 0,Y 311.685,Z 724.167,A -85,B 0,C 180,E1 14353.35,E2 14353.35} C_VEL
LIN {X 0,Y 306.075,Z 741.973,A -85,B 0,C 180,E1 14350.791,E2 14350.791} C_VEL
LIN {X 0,Y 300.589,Z 758.818,A -85,B 0,C 180,E1 14347.876,E2 14347.876} C_VEL
LIN {X 0,Y 295.535,Z 774.126,A -85,B 0,C 180,E1 14344.7,E2 14344.7} C_VEL
LIN {X 0,Y 290.977,Z 788.176,A -85,B 0,C 180,E1 14341.169,E2 14341.169} C_VEL
LIN {X 0,Y 287.323,Z 800.062,A -85,B 0,C 180,E1 14337.567,E2 14337.567} C_VEL
LIN {X 0,Y 284.347,Z 810.845,A -85,B 0,C 180,E1 14333.63,E2 14333.63} C_VEL
LIN {X 0,Y 282.298,Z 819.693,A -85,B 0,C 180,E1 14329.66,E2 14329.66} C_VEL
LIN {X 0,Y 281.064,Z 826.673,A -85,B 0,C 180,E1 14325.684,E2 14325.684} C_VEL
LIN {X 0,Y 280.478,Z 832.309,A -85,B 0,C 180,E1 14321.513,E2 14321.513} C_VEL
LIN {X 0,Y 280.386,Z 835.822,A -85,B 0,C 180,E1 14317.786,E2 14317.786} C_VEL
LIN {X 0,Y 280.479,Z 838.073,A -85,B 0,C 180,E1 14313.882,E2 14313.882} C_VEL
LIN {X 0,Y 280.555,Z 838.733,A -85,B 0,C 180,E1 14310.406,E2 14310.406} C_VEL
LIN {X 0,Y 280.509,Z 838.175,A -85,B 0,C 180,E1 14306.729,E2 14306.729} C_VEL
LIN {X 0,Y 280.409,Z 835.996,A -85,B 0,C 180,E1 14302.829,E2 14302.829} C_VEL
LIN {X 0,Y 280.461,Z 832.415,A -85,B 0,C 180,E1 14298.899,E2 14298.899} C_VEL
LIN {X 0,Y 280.963,Z 826.874,A -85,B 0,C 180,E1 14294.73,E2 14294.73} C_VEL
LIN {X 0,Y 282.218,Z 819.499,A -85,B 0,C 180,E1 14290.462,E2 14290.462} C_VEL
LIN {X 0,Y 284.305,Z 810.556,A -85,B 0,C 180,E1 14286.362,E2 14286.362} C_VEL
LIN {X 0,Y 287.467,Z 799.457,A -85,B 0,C 180,E1 14282.218,E2 14282.218} C_VEL
LIN {X 0,Y 291.785,Z 786.253,A -85,B 0,C 180,E1 14278.147,E2 14278.147} C_VEL
LIN {X 0,Y 297.035,Z 771.573,A -85,B 0,C 180,E1 14274.383,E2 14274.383} C_VEL
LIN {X 0,Y 303.464,Z 754.465,A -85,B 0,C 180,E1 14270.742,E2 14270.742} C_VEL
LIN {X 0,Y 310.666,Z 736.021,A -85,B 0,C 180,E1 14267.476,E2 14267.476} C_VEL
LIN {X 0,Y 319.056,Z 715.194,A -85,B 0,C 180,E1 14264.395,E2 14264.395} C_VEL
LIN {X 0,Y 328.738,Z 692.002,A -85,B 0,C 180,E1 14261.563,E2 14261.563} C_VEL
LIN {X 0,Y 339.222,Z 667.946,A -85,B 0,C 180,E1 14259.176,E2 14259.176} C_VEL
LIN {X 0,Y 349.284,Z 645.616,A -85,B 0,C 180,E1 14257.403,E2 14257.403} C_VEL
LIN {X 0,Y 356.209,Z 630.118,A -85,B 0,C 180,E1 14256.398,E2 14256.398} C_VEL
LIN {X 0,Y 346.15,Z 650.945,A -85,B 0,C 180,E1 14254.484,E2 14254.484} C_VEL
LIN {X 0,Y 335.971,Z 671.807,A -85,B 0,C 180,E1 14252.09,E2 14252.09} C_VEL
LIN {X 0,Y 326.435,Z 691.169,A -85,B 0,C 180,E1 14249.347,E2 14249.347} C_VEL
LIN {X 0,Y 317.746,Z 708.588,A -85,B 0,C 180,E1 14246.341,E2 14246.341} C_VEL
LIN {X 0,Y 309.721,Z 724.474,A -85,B 0,C 180,E1 14242.995,E2 14242.995} C_VEL
LIN {X 0,Y 302.751,Z 738.12,A -85,B 0,C 180,E1 14239.487,E2 14239.487} C_VEL
LIN {X 0,Y 296.56,Z 750.255,A -85,B 0,C 180,E1 14235.65,E2 14235.65} C_VEL
LIN {X 0,Y 291.487,Z 760.385,A -85,B 0,C 180,E1 14231.679,E2 14231.679} C_VEL
LIN {X 0,Y 287.349,Z 769.096,A -85,B 0,C 180,E1 14227.385,E2 14227.385} C_VEL
LIN {X 0,Y 284.49,Z 775.67,A -85,B 0,C 180,E1 14223.226,E2 14223.226} C_VEL
LIN {X 0,Y 282.543,Z 780.654,A -85,B 0,C 180,E1 14218.989,E2 14218.989} C_VEL
LIN {X 0,Y 281.389,Z 784.076,A -85,B 0,C 180,E1 14214.702,E2 14214.702} C_VEL
LIN {X 0,Y 280.798,Z 786.063,A -85,B 0,C 180,E1 14210.369,E2 14210.369} C_VEL
LIN {X 0,Y 280.592,Z 786.498,A -85,B 0,C 180,E1 14206.401,E2 14206.401} C_VEL
LIN {X 0,Y 280.548,Z 785.548,A -85,B 0,C 180,E1 14202.155,E2 14202.155} C_VEL
LIN {X 0,Y 280.704,Z 783.257,A -85,B 0,C 180,E1 14198.041,E2 14198.041} C_VEL
LIN {X 0,Y 281.212,Z 779.311,A -85,B 0,C 180,E1 14193.843,E2 14193.843} C_VEL
LIN {X 0,Y 282.296,Z 773.709,A -85,B 0,C 180,E1 14189.574,E2 14189.574} C_VEL
LIN {X 0,Y 284.087,Z 766.63,A -85,B 0,C 180,E1 14185.447,E2 14185.447} C_VEL
LIN {X 0,Y 286.708,Z 757.678,A -85,B 0,C 180,E1 14181.37,E2 14181.37} C_VEL
LIN {X 0,Y 290.092,Z 747.214,A -85,B 0,C 180,E1 14177.508,E2 14177.508} C_VEL
LIN {X 0,Y 294.289,Z 734.955,A -85,B 0,C 180,E1 14173.787,E2 14173.787} C_VEL
LIN {X 0,Y 299.095,Z 721.239,A -85,B 0,C 180,E1 14170.348,E2 14170.348} C_VEL
LIN {X 0,Y 304.319,Z 706.002,A -85,B 0,C 180,E1 14167.198,E2 14167.198} C_VEL
LIN {X 0,Y 309.677,Z 689.798,A -85,B 0,C 180,E1 14164.406,E2 14164.406} C_VEL
LIN {X 0,Y 315.316,Z 671.72,A -85,B 0,C 180,E1 14161.815,E2 14161.815} C_VEL
LIN {X 0,Y 320.752,Z 652.927,A -85,B 0,C 180,E1 14159.583,E2 14159.583} C_VEL
LIN {X 0,Y 326.031,Z 632.552,A -85,B 0,C 180,E1 14157.597,E2 14157.597} C_VEL
LIN {X 0,Y 330.743,Z 611.72,A -85,B 0,C 180,E1 14155.954,E2 14155.954} C_VEL
LIN {X 0,Y 334.953,Z 589.907,A -85,B 0,C 180,E1 14154.575,E2 14154.575} C_VEL
LIN {X 0,Y 338.512,Z 567.434,A -85,B 0,C 180,E1 14153.473,E2 14153.473} C_VEL
LIN {X 0,Y 341.288,Z 544.779,A -85,B 0,C 180,E1 14152.649,E2 14152.649} C_VEL
LIN {X 0,Y 355.169,Z 376.123,A -85,B 0,C 180,E1 14148.529,E2 14148.529} C_VEL
LIN {X 0,Y 343.133,Z 357.799,A -85,B 0,C 180,E1 14145.297,E2 14145.297} C_VEL
LIN {X 0,Y 332.184,Z 342.111,A -85,B 0,C 180,E1 14142.037,E2 14142.037} C_VEL
LIN {X 0,Y 322.51,Z 328.794,A -85,B 0,C 180,E1 14138.829,E2 14138.829} C_VEL
LIN {X 0,Y 314.405,Z 318.201,A -85,B 0,C 180,E1 14135.893,E2 14135.893} C_VEL
LIN {X 0,Y 310.209,Z 312.839,A -85,B 0,C 180,E1 14134.253,E2 14134.253} C_VEL
LIN {X 0,Y 306.254,Z 307.726,A -85,B 0,C 180,E1 14132.614,E2 14132.614} C_VEL
LIN {X 0,Y 302.82,Z 303.288,A -85,B 0,C 180,E1 14131.09,E2 14131.09} C_VEL
LIN {X 0,Y 298.408,Z 298.008,A -85,B 0,C 180,E1 14129.09,E2 14129.09} C_VEL
LIN {X 0,Y 297.362,Z 296.387,A -85,B 0,C 180,E1 14128.557,E2 14128.557} C_VEL
LIN {X 0,Y 294.134,Z 293.104,A -85,B 0,C 180,E1 14126.982,E2 14126.982} C_VEL
LIN {X 0,Y 292.502,Z 290.326,A -85,B 0,C 180,E1 14126.082,E2 14126.082} C_VEL
LIN {X 0,Y 289.394,Z 287.649,A -85,B 0,C 180,E1 14124.5,E2 14124.5} C_VEL
LIN {X 0,Y 287.359,Z 283.988,A -85,B 0,C 180,E1 14123.208,E2 14123.208} C_VEL
LIN {X 0,Y 284.242,Z 281.759,A -85,B 0,C 180,E1 14121.506,E2 14121.506} C_VEL
LIN {X 0,Y 282.609,Z 278.644,A -85,B 0,C 180,E1 14120.353,E2 14120.353} C_VEL
LIN {X 0,Y 282.386,Z 277.557,A -85,B 0,C 180,E1 14120.098,E2 14120.098} C_VEL
LIN {X 0,Y 282.381,Z 277.548,A -85,B 0,C 180,E1 14115.232,E2 14115.232} C_VEL
LIN {X 0,Y 282.401,Z 277.543,A -85,B 0,C 180,E1 14110.563,E2 14110.563} C_VEL
LIN {X 0,Y 282.384,Z 277.545,A -85,B 0,C 180,E1 14105.974,E2 14105.974} C_VEL
LIN {X 0,Y 282.372,Z 277.549,A -85,B 0,C 180,E1 14101.215,E2 14101.215} C_VEL
LIN {X 0,Y 282.395,Z 277.549,A -85,B 0,C 180,E1 14096.475,E2 14096.475} C_VEL
LIN {X 0,Y 282.379,Z 277.555,A -85,B 0,C 180,E1 14091.813,E2 14091.813} C_VEL
LIN {X 0,Y 282.365,Z 277.561,A -85,B 0,C 180,E1 14087.132,E2 14087.132} C_VEL
LIN {X 0,Y 282.378,Z 277.559,A -85,B 0,C 180,E1 14082.55,E2 14082.55} C_VEL
LIN {X 0,Y 282.396,Z 277.555,A -85,B 0,C 180,E1 14078.025,E2 14078.025} C_VEL
LIN {X 0,Y 282.364,Z 277.559,A -85,B 0,C 180,E1 14073.285,E2 14073.285} C_VEL
LIN {X 0,Y 282.366,Z 277.56,A -85,B 0,C 180,E1 14068.553,E2 14068.553} C_VEL
LIN {X 0,Y 282.358,Z 277.557,A -85,B 0,C 180,E1 14066.982,E2 14066.982} C_VEL
LIN {X 0,Y 281.484,Z 277.66,A -85,B 0,C 180,E1 14065.529,E2 14065.529} C_VEL
LIN {X 0,Y 277.831,Z 278.129,A -85,B 0,C 180,E1 14063.121,E2 14063.121} C_VEL
LIN {X 0,Y 274.772,Z 278.504,A -85,B 0,C 180,E1 14060.752,E2 14060.752} C_VEL
LIN {X 0,Y 274.442,Z 278.55,A -85,B 0,C 180,E1 14059.818,E2 14059.818} C_VEL
LIN {X 0,Y 274.415,Z 278.547,A -85,B 0,C 180,E1 14054.989,E2 14054.989} C_VEL
LIN {X 0,Y 274.422,Z 278.543,A -85,B 0,C 180,E1 14050.069,E2 14050.069} C_VEL
LIN {X 0,Y 274.433,Z 278.554,A -85,B 0,C 180,E1 14045.433,E2 14045.433} C_VEL
LIN {X 0,Y 274.433,Z 278.728,A -85,B 0,C 180,E1 14042.346,E2 14042.346} C_VEL
LIN {X 0,Y 275.495,Z 281.648,A -85,B 0,C 180,E1 14041.297,E2 14041.297} C_VEL
LIN {X 0,Y 277.956,Z 284.22,A -85,B 0,C 180,E1 14039.539,E2 14039.539} C_VEL
LIN {X 0,Y 279.872,Z 285.462,A -85,B 0,C 180,E1 14038.308,E2 14038.308} C_VEL
LIN {X 0,Y 281.583,Z 288.78,A -85,B 0,C 180,E1 14037.046,E2 14037.046} C_VEL
LIN {X 0,Y 284.737,Z 291.423,A -85,B 0,C 180,E1 14035.163,E2 14035.163} C_VEL
LIN {X 0,Y 288.003,Z 296.227,A -85,B 0,C 180,E1 14033.147,E2 14033.147} C_VEL
LIN {X 0,Y 289.719,Z 298.007,A -85,B 0,C 180,E1 14032.212,E2 14032.212} C_VEL
LIN {X 0,Y 293.921,Z 303.602,A -85,B 0,C 180,E1 14029.908,E2 14029.908} C_VEL
LIN {X 0,Y 298.478,Z 309.723,A -85,B 0,C 180,E1 14027.618,E2 14027.618} C_VEL
LIN {X 0,Y 305.698,Z 319.599,A -85,B 0,C 180,E1 14024.295,E2 14024.295} C_VEL
LIN {X 0,Y 315.473,Z 333.385,A -85,B 0,C 180,E1 14020.271,E2 14020.271} C_VEL
LIN {X 0,Y 325.903,Z 349.133,A -85,B 0,C 180,E1 14016.445,E2 14016.445} C_VEL
LIN {X 0,Y 336.202,Z 365.196,A -85,B 0,C 180,E1 14013.075,E2 14013.075} C_VEL
LIN {X 0,Y 347.297,Z 383.809,A -85,B 0,C 180,E1 14009.769,E2 14009.769} C_VEL
